   STATUS[239].EXT.Forced := FALSE;
   STATUS[239].EXT.BIT29 := FALSE;
   STATUS[239].EXT.BIT30 := FALSE;
   STATUS[239].EXT.BIT31 := FALSE;
   STATUS[239].EXT.ModeBit1 := FALSE;
   STATUS[239].EXT.ModeBit2 := FALSE;
   STATUS[239].EXT.ModeBit3 := FALSE;
   STATUS[239].EXT.BIT19 := FALSE;
   STATUS[239].EXT.BIT20 := FALSE;
   STATUS[239].EXT.AlarmSuppressed := FALSE;
   STATUS[239].EXT.AlarmPrsent := FALSE;
   STATUS[239].EXT.AlarmFailUnAck := FALSE;
   STATUS[239].Status := 0;
   STATUS[239].TimeStamp := 16#0000;
   STATUS[240].VALUE := 0.0;
   STATUS[240].TRIGVALUE := 0.0;
   STATUS[240].EXT.AlarmWarnUnAck := FALSE;
   STATUS[240].EXT.AckRequired := FALSE;
   STATUS[240].EXT.Maintanence := FALSE;
   STATUS[240].EXT.Operation := FALSE;
   STATUS[240].EXT.Forced := FALSE;
   STATUS[240].EXT.BIT29 := FALSE;
   STATUS[240].EXT.BIT30 := FALSE;
   STATUS[240].EXT.BIT31 := FALSE;
   STATUS[240].EXT.ModeBit1 := FALSE;
   STATUS[240].EXT.ModeBit2 := FALSE;
   STATUS[240].EXT.ModeBit3 := FALSE;
   STATUS[240].EXT.BIT19 := FALSE;
   STATUS[240].EXT.BIT20 := FALSE;
   STATUS[240].EXT.AlarmSuppressed := FALSE;
   STATUS[240].EXT.AlarmPrsent := FALSE;
   STATUS[240].EXT.AlarmFailUnAck := FALSE;
   STATUS[240].Status := 0;
   STATUS[240].TimeStamp := 16#0000;
   STATUS[241].VALUE := 0.0;
   STATUS[241].TRIGVALUE := 0.0;
   STATUS[241].EXT.AlarmWarnUnAck := FALSE;
   STATUS[241].EXT.AckRequired := FALSE;
   STATUS[241].EXT.Maintanence := FALSE;
   STATUS[241].EXT.Operation := FALSE;
   STATUS[241].EXT.Forced := FALSE;
   STATUS[241].EXT.BIT29 := FALSE;
   STATUS[241].EXT.BIT30 := FALSE;
   STATUS[241].EXT.BIT31 := FALSE;
   STATUS[241].EXT.ModeBit1 := FALSE;
   STATUS[241].EXT.ModeBit2 := FALSE;
   STATUS[241].EXT.ModeBit3 := FALSE;
   STATUS[241].EXT.BIT19 := FALSE;
   STATUS[241].EXT.BIT20 := FALSE;
   STATUS[241].EXT.AlarmSuppressed := FALSE;
   STATUS[241].EXT.AlarmPrsent := FALSE;
   STATUS[241].EXT.AlarmFailUnAck := FALSE;
   STATUS[241].Status := 0;
   STATUS[241].TimeStamp := 16#0000;
   STATUS[242].VALUE := 0.0;
   STATUS[242].TRIGVALUE := 0.0;
   STATUS[242].EXT.AlarmWarnUnAck := FALSE;
   STATUS[242].EXT.AckRequired := FALSE;
   STATUS[242].EXT.Maintanence := FALSE;
   STATUS[242].EXT.Operation := FALSE;
   STATUS[242].EXT.Forced := FALSE;
   STATUS[242].EXT.BIT29 := FALSE;
   STATUS[242].EXT.BIT30 := FALSE;
   STATUS[242].EXT.BIT31 := FALSE;
   STATUS[242].EXT.ModeBit1 := FALSE;
   STATUS[242].EXT.ModeBit2 := FALSE;
   STATUS[242].EXT.ModeBit3 := FALSE;
   STATUS[242].EXT.BIT19 := FALSE;
   STATUS[242].EXT.BIT20 := FALSE;
   STATUS[242].EXT.AlarmSuppressed := FALSE;
   STATUS[242].EXT.AlarmPrsent := FALSE;
   STATUS[242].EXT.AlarmFailUnAck := FALSE;
   STATUS[242].Status := 0;
   STATUS[242].TimeStamp := 16#0000;
   STATUS[243].VALUE := 0.0;
   STATUS[243].TRIGVALUE := 0.0;
   STATUS[243].EXT.AlarmWarnUnAck := FALSE;
   STATUS[243].EXT.AckRequired := FALSE;
   STATUS[243].EXT.Maintanence := FALSE;
   STATUS[243].EXT.Operation := FALSE;
   STATUS[243].EXT.Forced := FALSE;
   STATUS[243].EXT.BIT29 := FALSE;
   STATUS[243].EXT.BIT30 := FALSE;
   STATUS[243].EXT.BIT31 := FALSE;
   STATUS[243].EXT.ModeBit1 := FALSE;
   STATUS[243].EXT.ModeBit2 := FALSE;
   STATUS[243].EXT.ModeBit3 := FALSE;
   STATUS[243].EXT.BIT19 := FALSE;
   STATUS[243].EXT.BIT20 := FALSE;
   STATUS[243].EXT.AlarmSuppressed := FALSE;
   STATUS[243].EXT.AlarmPrsent := FALSE;
   STATUS[243].EXT.AlarmFailUnAck := FALSE;
   STATUS[243].Status := 0;
   STATUS[243].TimeStamp := 16#0000;
   STATUS[244].VALUE := 0.0;
   STATUS[244].TRIGVALUE := 0.0;
   STATUS[244].EXT.AlarmWarnUnAck := FALSE;
   STATUS[244].EXT.AckRequired := FALSE;
   STATUS[244].EXT.Maintanence := FALSE;
   STATUS[244].EXT.Operation := FALSE;
   STATUS[244].EXT.Forced := FALSE;
   STATUS[244].EXT.BIT29 := FALSE;
   STATUS[244].EXT.BIT30 := FALSE;
   STATUS[244].EXT.BIT31 := FALSE;
   STATUS[244].EXT.ModeBit1 := FALSE;
   STATUS[244].EXT.ModeBit2 := FALSE;
   STATUS[244].EXT.ModeBit3 := FALSE;
   STATUS[244].EXT.BIT19 := FALSE;
   STATUS[244].EXT.BIT20 := FALSE;
   STATUS[244].EXT.AlarmSuppressed := FALSE;
   STATUS[244].EXT.AlarmPrsent := FALSE;
   STATUS[244].EXT.AlarmFailUnAck := FALSE;
   STATUS[244].Status := 0;
   STATUS[244].TimeStamp := 16#0000;
   STATUS[245].VALUE := 0.0;
   STATUS[245].TRIGVALUE := 0.0;
   STATUS[245].EXT.AlarmWarnUnAck := FALSE;
   STATUS[245].EXT.AckRequired := FALSE;
   STATUS[245].EXT.Maintanence := FALSE;
   STATUS[245].EXT.Operation := FALSE;
   STATUS[245].EXT.Forced := FALSE;
   STATUS[245].EXT.BIT29 := FALSE;
   STATUS[245].EXT.BIT30 := FALSE;
   STATUS[245].EXT.BIT31 := FALSE;
   STATUS[245].EXT.ModeBit1 := FALSE;
   STATUS[245].EXT.ModeBit2 := FALSE;
   STATUS[245].EXT.ModeBit3 := FALSE;
   STATUS[245].EXT.BIT19 := FALSE;
   STATUS[245].EXT.BIT20 := FALSE;
   STATUS[245].EXT.AlarmSuppressed := FALSE;
   STATUS[245].EXT.AlarmPrsent := FALSE;
   STATUS[245].EXT.AlarmFailUnAck := FALSE;
   STATUS[245].Status := 0;
   STATUS[245].TimeStamp := 16#0000;
   STATUS[246].VALUE := 0.0;
   STATUS[246].TRIGVALUE := 0.0;
   STATUS[246].EXT.AlarmWarnUnAck := FALSE;
   STATUS[246].EXT.AckRequired := FALSE;
   STATUS[246].EXT.Maintanence := FALSE;
   STATUS[246].EXT.Operation := FALSE;
   STATUS[246].EXT.Forced := FALSE;
   STATUS[246].EXT.BIT29 := FALSE;
   STATUS[246].EXT.BIT30 := FALSE;
   STATUS[246].EXT.BIT31 := FALSE;
   STATUS[246].EXT.ModeBit1 := FALSE;
   STATUS[246].EXT.ModeBit2 := FALSE;
   STATUS[246].EXT.ModeBit3 := FALSE;
   STATUS[246].EXT.BIT19 := FALSE;
   STATUS[246].EXT.BIT20 := FALSE;
   STATUS[246].EXT.AlarmSuppressed := FALSE;
   STATUS[246].EXT.AlarmPrsent := FALSE;
   STATUS[246].EXT.AlarmFailUnAck := FALSE;
   STATUS[246].Status := 0;
   STATUS[246].TimeStamp := 16#0000;
   STATUS[247].VALUE := 0.0;
   STATUS[247].TRIGVALUE := 0.0;
   STATUS[247].EXT.AlarmWarnUnAck := FALSE;
   STATUS[247].EXT.AckRequired := FALSE;
   STATUS[247].EXT.Maintanence := FALSE;
   STATUS[247].EXT.Operation := FALSE;
   STATUS[247].EXT.Forced := FALSE;
   STATUS[247].EXT.BIT29 := FALSE;
   STATUS[247].EXT.BIT30 := FALSE;
   STATUS[247].EXT.BIT31 := FALSE;
   STATUS[247].EXT.ModeBit1 := FALSE;
   STATUS[247].EXT.ModeBit2 := FALSE;
   STATUS[247].EXT.ModeBit3 := FALSE;
   STATUS[247].EXT.BIT19 := FALSE;
   STATUS[247].EXT.BIT20 := FALSE;
   STATUS[247].EXT.AlarmSuppressed := FALSE;
   STATUS[247].EXT.AlarmPrsent := FALSE;
   STATUS[247].EXT.AlarmFailUnAck := FALSE;
   STATUS[247].Status := 0;
   STATUS[247].TimeStamp := 16#0000;
   STATUS[248].VALUE := 0.0;
   STATUS[248].TRIGVALUE := 0.0;
   STATUS[248].EXT.AlarmWarnUnAck := FALSE;
   STATUS[248].EXT.AckRequired := FALSE;
   STATUS[248].EXT.Maintanence := FALSE;
   STATUS[248].EXT.Operation := FALSE;
   STATUS[248].EXT.Forced := FALSE;
   STATUS[248].EXT.BIT29 := FALSE;
   STATUS[248].EXT.BIT30 := FALSE;
   STATUS[248].EXT.BIT31 := FALSE;
   STATUS[248].EXT.ModeBit1 := FALSE;
   STATUS[248].EXT.ModeBit2 := FALSE;
   STATUS[248].EXT.ModeBit3 := FALSE;
   STATUS[248].EXT.BIT19 := FALSE;
   STATUS[248].EXT.BIT20 := FALSE;
   STATUS[248].EXT.AlarmSuppressed := FALSE;
   STATUS[248].EXT.AlarmPrsent := FALSE;
   STATUS[248].EXT.AlarmFailUnAck := FALSE;
   STATUS[248].Status := 0;
   STATUS[248].TimeStamp := 16#0000;
   STATUS[249].VALUE := 0.0;
   STATUS[249].TRIGVALUE := 0.0;
   STATUS[249].EXT.AlarmWarnUnAck := FALSE;
   STATUS[249].EXT.AckRequired := FALSE;
   STATUS[249].EXT.Maintanence := FALSE;
   STATUS[249].EXT.Operation := FALSE;
   STATUS[249].EXT.Forced := FALSE;
   STATUS[249].EXT.BIT29 := FALSE;
   STATUS[249].EXT.BIT30 := FALSE;
   STATUS[249].EXT.BIT31 := FALSE;
   STATUS[249].EXT.ModeBit1 := FALSE;
   STATUS[249].EXT.ModeBit2 := FALSE;
   STATUS[249].EXT.ModeBit3 := FALSE;
   STATUS[249].EXT.BIT19 := FALSE;
   STATUS[249].EXT.BIT20 := FALSE;
   STATUS[249].EXT.AlarmSuppressed := FALSE;
   STATUS[249].EXT.AlarmPrsent := FALSE;
   STATUS[249].EXT.AlarmFailUnAck := FALSE;
   STATUS[249].Status := 0;
   STATUS[249].TimeStamp := 16#0000;
   STATUS[250].VALUE := 0.0;
   STATUS[250].TRIGVALUE := 0.0;
   STATUS[250].EXT.AlarmWarnUnAck := FALSE;
   STATUS[250].EXT.AckRequired := FALSE;
   STATUS[250].EXT.Maintanence := FALSE;
   STATUS[250].EXT.Operation := FALSE;
   STATUS[250].EXT.Forced := FALSE;
   STATUS[250].EXT.BIT29 := FALSE;
   STATUS[250].EXT.BIT30 := FALSE;
   STATUS[250].EXT.BIT31 := FALSE;
   STATUS[250].EXT.ModeBit1 := FALSE;
   STATUS[250].EXT.ModeBit2 := FALSE;
   STATUS[250].EXT.ModeBit3 := FALSE;
   STATUS[250].EXT.BIT19 := FALSE;
   STATUS[250].EXT.BIT20 := FALSE;
   STATUS[250].EXT.AlarmSuppressed := FALSE;
   STATUS[250].EXT.AlarmPrsent := FALSE;
   STATUS[250].EXT.AlarmFailUnAck := FALSE;
   STATUS[250].Status := 0;
   STATUS[250].TimeStamp := 16#0000;
   STATUS[251].VALUE := 0.0;
   STATUS[251].TRIGVALUE := 0.0;
   STATUS[251].EXT.AlarmWarnUnAck := FALSE;
   STATUS[251].EXT.AckRequired := FALSE;
   STATUS[251].EXT.Maintanence := FALSE;
   STATUS[251].EXT.Operation := FALSE;
   STATUS[251].EXT.Forced := FALSE;
   STATUS[251].EXT.BIT29 := FALSE;
   STATUS[251].EXT.BIT30 := FALSE;
   STATUS[251].EXT.BIT31 := FALSE;
   STATUS[251].EXT.ModeBit1 := FALSE;
   STATUS[251].EXT.ModeBit2 := FALSE;
   STATUS[251].EXT.ModeBit3 := FALSE;
   STATUS[251].EXT.BIT19 := FALSE;
   STATUS[251].EXT.BIT20 := FALSE;
   STATUS[251].EXT.AlarmSuppressed := FALSE;
   STATUS[251].EXT.AlarmPrsent := FALSE;
   STATUS[251].EXT.AlarmFailUnAck := FALSE;
   STATUS[251].Status := 0;
   STATUS[251].TimeStamp := 16#0000;
   STATUS[252].VALUE := 0.0;
   STATUS[252].TRIGVALUE := 0.0;
   STATUS[252].EXT.AlarmWarnUnAck := FALSE;
   STATUS[252].EXT.AckRequired := FALSE;
   STATUS[252].EXT.Maintanence := FALSE;
   STATUS[252].EXT.Operation := FALSE;
   STATUS[252].EXT.Forced := FALSE;
   STATUS[252].EXT.BIT29 := FALSE;
   STATUS[252].EXT.BIT30 := FALSE;
   STATUS[252].EXT.BIT31 := FALSE;
   STATUS[252].EXT.ModeBit1 := FALSE;
   STATUS[252].EXT.ModeBit2 := FALSE;
   STATUS[252].EXT.ModeBit3 := FALSE;
   STATUS[252].EXT.BIT19 := FALSE;
   STATUS[252].EXT.BIT20 := FALSE;
   STATUS[252].EXT.AlarmSuppressed := FALSE;
   STATUS[252].EXT.AlarmPrsent := FALSE;
   STATUS[252].EXT.AlarmFailUnAck := FALSE;
   STATUS[252].Status := 0;
   STATUS[252].TimeStamp := 16#0000;
   STATUS[253].VALUE := 0.0;
   STATUS[253].TRIGVALUE := 0.0;
   STATUS[253].EXT.AlarmWarnUnAck := FALSE;
   STATUS[253].EXT.AckRequired := FALSE;
   STATUS[253].EXT.Maintanence := FALSE;
   STATUS[253].EXT.Operation := FALSE;
   STATUS[253].EXT.Forced := FALSE;
   STATUS[253].EXT.BIT29 := FALSE;
   STATUS[253].EXT.BIT30 := FALSE;
   STATUS[253].EXT.BIT31 := FALSE;
   STATUS[253].EXT.ModeBit1 := FALSE;
   STATUS[253].EXT.ModeBit2 := FALSE;
   STATUS[253].EXT.ModeBit3 := FALSE;
   STATUS[253].EXT.BIT19 := FALSE;
   STATUS[253].EXT.BIT20 := FALSE;
   STATUS[253].EXT.AlarmSuppressed := FALSE;
   STATUS[253].EXT.AlarmPrsent := FALSE;
   STATUS[253].EXT.AlarmFailUnAck := FALSE;
   STATUS[253].Status := 0;
   STATUS[253].TimeStamp := 16#0000;
   STATUS[254].VALUE := 0.0;
   STATUS[254].TRIGVALUE := 0.0;
   STATUS[254].EXT.AlarmWarnUnAck := FALSE;
   STATUS[254].EXT.AckRequired := FALSE;
   STATUS[254].EXT.Maintanence := FALSE;
   STATUS[254].EXT.Operation := FALSE;
   STATUS[254].EXT.Forced := FALSE;
   STATUS[254].EXT.BIT29 := FALSE;
   STATUS[254].EXT.BIT30 := FALSE;
   STATUS[254].EXT.BIT31 := FALSE;
   STATUS[254].EXT.ModeBit1 := FALSE;
   STATUS[254].EXT.ModeBit2 := FALSE;
   STATUS[254].EXT.ModeBit3 := FALSE;
   STATUS[254].EXT.BIT19 := FALSE;
   STATUS[254].EXT.BIT20 := FALSE;
   STATUS[254].EXT.AlarmSuppressed := FALSE;
   STATUS[254].EXT.AlarmPrsent := FALSE;
   STATUS[254].EXT.AlarmFailUnAck := FALSE;
   STATUS[254].Status := 0;
   STATUS[254].TimeStamp := 16#0000;
   STATUS[255].VALUE := 0.0;
   STATUS[255].TRIGVALUE := 0.0;
   STATUS[255].EXT.AlarmWarnUnAck := FALSE;
   STATUS[255].EXT.AckRequired := FALSE;
   STATUS[255].EXT.Maintanence := FALSE;
   STATUS[255].EXT.Operation := FALSE;
   STATUS[255].EXT.Forced := FALSE;
   STATUS[255].EXT.BIT29 := FALSE;
   STATUS[255].EXT.BIT30 := FALSE;
   STATUS[255].EXT.BIT31 := FALSE;
   STATUS[255].EXT.ModeBit1 := FALSE;
   STATUS[255].EXT.ModeBit2 := FALSE;
   STATUS[255].EXT.ModeBit3 := FALSE;
   STATUS[255].EXT.BIT19 := FALSE;
   STATUS[255].EXT.BIT20 := FALSE;
   STATUS[255].EXT.AlarmSuppressed := FALSE;
   STATUS[255].EXT.AlarmPrsent := FALSE;
   STATUS[255].EXT.AlarmFailUnAck := FALSE;
   STATUS[255].Status := 0;
   STATUS[255].TimeStamp := 16#0000;
   STATUS[256].VALUE := 0.0;
   STATUS[256].TRIGVALUE := 0.0;
   STATUS[256].EXT.AlarmWarnUnAck := FALSE;
   STATUS[256].EXT.AckRequired := FALSE;
   STATUS[256].EXT.Maintanence := FALSE;
   STATUS[256].EXT.Operation := FALSE;
   STATUS[256].EXT.Forced := FALSE;
   STATUS[256].EXT.BIT29 := FALSE;
   STATUS[256].EXT.BIT30 := FALSE;
   STATUS[256].EXT.BIT31 := FALSE;
   STATUS[256].EXT.ModeBit1 := FALSE;
   STATUS[256].EXT.ModeBit2 := FALSE;
   STATUS[256].EXT.ModeBit3 := FALSE;
   STATUS[256].EXT.BIT19 := FALSE;
   STATUS[256].EXT.BIT20 := FALSE;
   STATUS[256].EXT.AlarmSuppressed := FALSE;
   STATUS[256].EXT.AlarmPrsent := FALSE;
   STATUS[256].EXT.AlarmFailUnAck := FALSE;
   STATUS[256].Status := 0;
   STATUS[256].TimeStamp := 16#0000;
   STATUS[257].VALUE := 0.0;
   STATUS[257].TRIGVALUE := 0.0;
   STATUS[257].EXT.AlarmWarnUnAck := FALSE;
   STATUS[257].EXT.AckRequired := FALSE;
   STATUS[257].EXT.Maintanence := FALSE;
   STATUS[257].EXT.Operation := FALSE;
   STATUS[257].EXT.Forced := FALSE;
   STATUS[257].EXT.BIT29 := FALSE;
   STATUS[257].EXT.BIT30 := FALSE;
   STATUS[257].EXT.BIT31 := FALSE;
   STATUS[257].EXT.ModeBit1 := FALSE;
   STATUS[257].EXT.ModeBit2 := FALSE;
   STATUS[257].EXT.ModeBit3 := FALSE;
   STATUS[257].EXT.BIT19 := FALSE;
   STATUS[257].EXT.BIT20 := FALSE;
   STATUS[257].EXT.AlarmSuppressed := FALSE;
   STATUS[257].EXT.AlarmPrsent := FALSE;
   STATUS[257].EXT.AlarmFailUnAck := FALSE;
   STATUS[257].Status := 0;
   STATUS[257].TimeStamp := 16#0000;
   STATUS[258].VALUE := 0.0;
   STATUS[258].TRIGVALUE := 0.0;
   STATUS[258].EXT.AlarmWarnUnAck := FALSE;
   STATUS[258].EXT.AckRequired := FALSE;
   STATUS[258].EXT.Maintanence := FALSE;
   STATUS[258].EXT.Operation := FALSE;
   STATUS[258].EXT.Forced := FALSE;
   STATUS[258].EXT.BIT29 := FALSE;
   STATUS[258].EXT.BIT30 := FALSE;
   STATUS[258].EXT.BIT31 := FALSE;
   STATUS[258].EXT.ModeBit1 := FALSE;
   STATUS[258].EXT.ModeBit2 := FALSE;
   STATUS[258].EXT.ModeBit3 := FALSE;
   STATUS[258].EXT.BIT19 := FALSE;
   STATUS[258].EXT.BIT20 := FALSE;
   STATUS[258].EXT.AlarmSuppressed := FALSE;
   STATUS[258].EXT.AlarmPrsent := FALSE;
   STATUS[258].EXT.AlarmFailUnAck := FALSE;
   STATUS[258].Status := 0;
   STATUS[258].TimeStamp := 16#0000;
   STATUS[259].VALUE := 0.0;
   STATUS[259].TRIGVALUE := 0.0;
   STATUS[259].EXT.AlarmWarnUnAck := FALSE;
   STATUS[259].EXT.AckRequired := FALSE;
   STATUS[259].EXT.Maintanence := FALSE;
   STATUS[259].EXT.Operation := FALSE;
   STATUS[259].EXT.Forced := FALSE;
   STATUS[259].EXT.BIT29 := FALSE;
   STATUS[259].EXT.BIT30 := FALSE;
   STATUS[259].EXT.BIT31 := FALSE;
   STATUS[259].EXT.ModeBit1 := FALSE;
   STATUS[259].EXT.ModeBit2 := FALSE;
   STATUS[259].EXT.ModeBit3 := FALSE;
   STATUS[259].EXT.BIT19 := FALSE;
   STATUS[259].EXT.BIT20 := FALSE;
   STATUS[259].EXT.AlarmSuppressed := FALSE;
   STATUS[259].EXT.AlarmPrsent := FALSE;
   STATUS[259].EXT.AlarmFailUnAck := FALSE;
   STATUS[259].Status := 0;
   STATUS[259].TimeStamp := 16#0000;
   STATUS[260].VALUE := 0.0;
   STATUS[260].TRIGVALUE := 0.0;
   STATUS[260].EXT.AlarmWarnUnAck := FALSE;
   STATUS[260].EXT.AckRequired := FALSE;
   STATUS[260].EXT.Maintanence := FALSE;
   STATUS[260].EXT.Operation := FALSE;
   STATUS[260].EXT.Forced := FALSE;
   STATUS[260].EXT.BIT29 := FALSE;
   STATUS[260].EXT.BIT30 := FALSE;
   STATUS[260].EXT.BIT31 := FALSE;
   STATUS[260].EXT.ModeBit1 := FALSE;
   STATUS[260].EXT.ModeBit2 := FALSE;
   STATUS[260].EXT.ModeBit3 := FALSE;
   STATUS[260].EXT.BIT19 := FALSE;
   STATUS[260].EXT.BIT20 := FALSE;
   STATUS[260].EXT.AlarmSuppressed := FALSE;
   STATUS[260].EXT.AlarmPrsent := FALSE;
   STATUS[260].EXT.AlarmFailUnAck := FALSE;
   STATUS[260].Status := 0;
   STATUS[260].TimeStamp := 16#0000;
   STATUS[261].VALUE := 0.0;
   STATUS[261].TRIGVALUE := 0.0;
   STATUS[261].EXT.AlarmWarnUnAck := FALSE;
   STATUS[261].EXT.AckRequired := FALSE;
   STATUS[261].EXT.Maintanence := FALSE;
   STATUS[261].EXT.Operation := FALSE;
   STATUS[261].EXT.Forced := FALSE;
   STATUS[261].EXT.BIT29 := FALSE;
   STATUS[261].EXT.BIT30 := FALSE;
   STATUS[261].EXT.BIT31 := FALSE;
   STATUS[261].EXT.ModeBit1 := FALSE;
   STATUS[261].EXT.ModeBit2 := FALSE;
   STATUS[261].EXT.ModeBit3 := FALSE;
   STATUS[261].EXT.BIT19 := FALSE;
   STATUS[261].EXT.BIT20 := FALSE;
   STATUS[261].EXT.AlarmSuppressed := FALSE;
   STATUS[261].EXT.AlarmPrsent := FALSE;
   STATUS[261].EXT.AlarmFailUnAck := FALSE;
   STATUS[261].Status := 0;
   STATUS[261].TimeStamp := 16#0000;
   STATUS[262].VALUE := 0.0;
   STATUS[262].TRIGVALUE := 0.0;
   STATUS[262].EXT.AlarmWarnUnAck := FALSE;
   STATUS[262].EXT.AckRequired := FALSE;
   STATUS[262].EXT.Maintanence := FALSE;
   STATUS[262].EXT.Operation := FALSE;
   STATUS[262].EXT.Forced := FALSE;
   STATUS[262].EXT.BIT29 := FALSE;
   STATUS[262].EXT.BIT30 := FALSE;
   STATUS[262].EXT.BIT31 := FALSE;
   STATUS[262].EXT.ModeBit1 := FALSE;
   STATUS[262].EXT.ModeBit2 := FALSE;
   STATUS[262].EXT.ModeBit3 := FALSE;
   STATUS[262].EXT.BIT19 := FALSE;
   STATUS[262].EXT.BIT20 := FALSE;
   STATUS[262].EXT.AlarmSuppressed := FALSE;
   STATUS[262].EXT.AlarmPrsent := FALSE;
   STATUS[262].EXT.AlarmFailUnAck := FALSE;
   STATUS[262].Status := 0;
   STATUS[262].TimeStamp := 16#0000;
   STATUS[263].VALUE := 0.0;
   STATUS[263].TRIGVALUE := 0.0;
   STATUS[263].EXT.AlarmWarnUnAck := FALSE;
   STATUS[263].EXT.AckRequired := FALSE;
   STATUS[263].EXT.Maintanence := FALSE;
   STATUS[263].EXT.Operation := FALSE;
   STATUS[263].EXT.Forced := FALSE;
   STATUS[263].EXT.BIT29 := FALSE;
   STATUS[263].EXT.BIT30 := FALSE;
   STATUS[263].EXT.BIT31 := FALSE;
   STATUS[263].EXT.ModeBit1 := FALSE;
   STATUS[263].EXT.ModeBit2 := FALSE;
   STATUS[263].EXT.ModeBit3 := FALSE;
   STATUS[263].EXT.BIT19 := FALSE;
   STATUS[263].EXT.BIT20 := FALSE;
   STATUS[263].EXT.AlarmSuppressed := FALSE;
   STATUS[263].EXT.AlarmPrsent := FALSE;
   STATUS[263].EXT.AlarmFailUnAck := FALSE;
   STATUS[263].Status := 0;
   STATUS[263].TimeStamp := 16#0000;
   STATUS[264].VALUE := 0.0;
   STATUS[264].TRIGVALUE := 0.0;
   STATUS[264].EXT.AlarmWarnUnAck := FALSE;
   STATUS[264].EXT.AckRequired := FALSE;
   STATUS[264].EXT.Maintanence := FALSE;
   STATUS[264].EXT.Operation := FALSE;
   STATUS[264].EXT.Forced := FALSE;
   STATUS[264].EXT.BIT29 := FALSE;
   STATUS[264].EXT.BIT30 := FALSE;
   STATUS[264].EXT.BIT31 := FALSE;
   STATUS[264].EXT.ModeBit1 := FALSE;
   STATUS[264].EXT.ModeBit2 := FALSE;
   STATUS[264].EXT.ModeBit3 := FALSE;
   STATUS[264].EXT.BIT19 := FALSE;
   STATUS[264].EXT.BIT20 := FALSE;
   STATUS[264].EXT.AlarmSuppressed := FALSE;
   STATUS[264].EXT.AlarmPrsent := FALSE;
   STATUS[264].EXT.AlarmFailUnAck := FALSE;
   STATUS[264].Status := 0;
   STATUS[264].TimeStamp := 16#0000;
   STATUS[265].VALUE := 0.0;
   STATUS[265].TRIGVALUE := 0.0;
   STATUS[265].EXT.AlarmWarnUnAck := FALSE;
   STATUS[265].EXT.AckRequired := FALSE;
   STATUS[265].EXT.Maintanence := FALSE;
   STATUS[265].EXT.Operation := FALSE;
   STATUS[265].EXT.Forced := FALSE;
   STATUS[265].EXT.BIT29 := FALSE;
   STATUS[265].EXT.BIT30 := FALSE;
   STATUS[265].EXT.BIT31 := FALSE;
   STATUS[265].EXT.ModeBit1 := FALSE;
   STATUS[265].EXT.ModeBit2 := FALSE;
   STATUS[265].EXT.ModeBit3 := FALSE;
   STATUS[265].EXT.BIT19 := FALSE;
   STATUS[265].EXT.BIT20 := FALSE;
   STATUS[265].EXT.AlarmSuppressed := FALSE;
   STATUS[265].EXT.AlarmPrsent := FALSE;
   STATUS[265].EXT.AlarmFailUnAck := FALSE;
   STATUS[265].Status := 0;
   STATUS[265].TimeStamp := 16#0000;
   STATUS[266].VALUE := 0.0;
   STATUS[266].TRIGVALUE := 0.0;
   STATUS[266].EXT.AlarmWarnUnAck := FALSE;
   STATUS[266].EXT.AckRequired := FALSE;
   STATUS[266].EXT.Maintanence := FALSE;
   STATUS[266].EXT.Operation := FALSE;
   STATUS[266].EXT.Forced := FALSE;
   STATUS[266].EXT.BIT29 := FALSE;
   STATUS[266].EXT.BIT30 := FALSE;
   STATUS[266].EXT.BIT31 := FALSE;
   STATUS[266].EXT.ModeBit1 := FALSE;
   STATUS[266].EXT.ModeBit2 := FALSE;
   STATUS[266].EXT.ModeBit3 := FALSE;
   STATUS[266].EXT.BIT19 := FALSE;
   STATUS[266].EXT.BIT20 := FALSE;
   STATUS[266].EXT.AlarmSuppressed := FALSE;
   STATUS[266].EXT.AlarmPrsent := FALSE;
   STATUS[266].EXT.AlarmFailUnAck := FALSE;
   STATUS[266].Status := 0;
   STATUS[266].TimeStamp := 16#0000;
   STATUS[267].VALUE := 0.0;
   STATUS[267].TRIGVALUE := 0.0;
   STATUS[267].EXT.AlarmWarnUnAck := FALSE;
   STATUS[267].EXT.AckRequired := FALSE;
   STATUS[267].EXT.Maintanence := FALSE;
   STATUS[267].EXT.Operation := FALSE;
   STATUS[267].EXT.Forced := FALSE;
   STATUS[267].EXT.BIT29 := FALSE;
   STATUS[267].EXT.BIT30 := FALSE;
   STATUS[267].EXT.BIT31 := FALSE;
   STATUS[267].EXT.ModeBit1 := FALSE;
   STATUS[267].EXT.ModeBit2 := FALSE;
   STATUS[267].EXT.ModeBit3 := FALSE;
   STATUS[267].EXT.BIT19 := FALSE;
   STATUS[267].EXT.BIT20 := FALSE;
   STATUS[267].EXT.AlarmSuppressed := FALSE;
   STATUS[267].EXT.AlarmPrsent := FALSE;
   STATUS[267].EXT.AlarmFailUnAck := FALSE;
   STATUS[267].Status := 0;
   STATUS[267].TimeStamp := 16#0000;
   STATUS[268].VALUE := 0.0;
   STATUS[268].TRIGVALUE := 0.0;
   STATUS[268].EXT.AlarmWarnUnAck := FALSE;
   STATUS[268].EXT.AckRequired := FALSE;
   STATUS[268].EXT.Maintanence := FALSE;
   STATUS[268].EXT.Operation := FALSE;
   STATUS[268].EXT.Forced := FALSE;
   STATUS[268].EXT.BIT29 := FALSE;
   STATUS[268].EXT.BIT30 := FALSE;
   STATUS[268].EXT.BIT31 := FALSE;
   STATUS[268].EXT.ModeBit1 := FALSE;
   STATUS[268].EXT.ModeBit2 := FALSE;
   STATUS[268].EXT.ModeBit3 := FALSE;
   STATUS[268].EXT.BIT19 := FALSE;
   STATUS[268].EXT.BIT20 := FALSE;
   STATUS[268].EXT.AlarmSuppressed := FALSE;
   STATUS[268].EXT.AlarmPrsent := FALSE;
   STATUS[268].EXT.AlarmFailUnAck := FALSE;
   STATUS[268].Status := 0;
   STATUS[268].TimeStamp := 16#0000;
   STATUS[269].VALUE := 0.0;
   STATUS[269].TRIGVALUE := 0.0;
   STATUS[269].EXT.AlarmWarnUnAck := FALSE;
   STATUS[269].EXT.AckRequired := FALSE;
   STATUS[269].EXT.Maintanence := FALSE;
   STATUS[269].EXT.Operation := FALSE;
   STATUS[269].EXT.Forced := FALSE;
   STATUS[269].EXT.BIT29 := FALSE;
   STATUS[269].EXT.BIT30 := FALSE;
   STATUS[269].EXT.BIT31 := FALSE;
   STATUS[269].EXT.ModeBit1 := FALSE;
   STATUS[269].EXT.ModeBit2 := FALSE;
   STATUS[269].EXT.ModeBit3 := FALSE;
   STATUS[269].EXT.BIT19 := FALSE;
   STATUS[269].EXT.BIT20 := FALSE;
   STATUS[269].EXT.AlarmSuppressed := FALSE;
   STATUS[269].EXT.AlarmPrsent := FALSE;
   STATUS[269].EXT.AlarmFailUnAck := FALSE;
   STATUS[269].Status := 0;
   STATUS[269].TimeStamp := 16#0000;
   STATUS[270].VALUE := 0.0;
   STATUS[270].TRIGVALUE := 0.0;
   STATUS[270].EXT.AlarmWarnUnAck := FALSE;
   STATUS[270].EXT.AckRequired := FALSE;
   STATUS[270].EXT.Maintanence := FALSE;
   STATUS[270].EXT.Operation := FALSE;
   STATUS[270].EXT.Forced := FALSE;
   STATUS[270].EXT.BIT29 := FALSE;
   STATUS[270].EXT.BIT30 := FALSE;
   STATUS[270].EXT.BIT31 := FALSE;
   STATUS[270].EXT.ModeBit1 := FALSE;
   STATUS[270].EXT.ModeBit2 := FALSE;
   STATUS[270].EXT.ModeBit3 := FALSE;
   STATUS[270].EXT.BIT19 := FALSE;
   STATUS[270].EXT.BIT20 := FALSE;
   STATUS[270].EXT.AlarmSuppressed := FALSE;
   STATUS[270].EXT.AlarmPrsent := FALSE;
   STATUS[270].EXT.AlarmFailUnAck := FALSE;
   STATUS[270].Status := 0;
   STATUS[270].TimeStamp := 16#0000;
   STATUS[271].VALUE := 0.0;
   STATUS[271].TRIGVALUE := 0.0;
   STATUS[271].EXT.AlarmWarnUnAck := FALSE;
   STATUS[271].EXT.AckRequired := FALSE;
   STATUS[271].EXT.Maintanence := FALSE;
   STATUS[271].EXT.Operation := FALSE;
   STATUS[271].EXT.Forced := FALSE;
   STATUS[271].EXT.BIT29 := FALSE;
   STATUS[271].EXT.BIT30 := FALSE;
   STATUS[271].EXT.BIT31 := FALSE;
   STATUS[271].EXT.ModeBit1 := FALSE;
   STATUS[271].EXT.ModeBit2 := FALSE;
   STATUS[271].EXT.ModeBit3 := FALSE;
   STATUS[271].EXT.BIT19 := FALSE;
   STATUS[271].EXT.BIT20 := FALSE;
   STATUS[271].EXT.AlarmSuppressed := FALSE;
   STATUS[271].EXT.AlarmPrsent := FALSE;
   STATUS[271].EXT.AlarmFailUnAck := FALSE;
   STATUS[271].Status := 0;
   STATUS[271].TimeStamp := 16#0000;
   STATUS[272].VALUE := 0.0;
   STATUS[272].TRIGVALUE := 0.0;
   STATUS[272].EXT.AlarmWarnUnAck := FALSE;
   STATUS[272].EXT.AckRequired := FALSE;
   STATUS[272].EXT.Maintanence := FALSE;
   STATUS[272].EXT.Operation := FALSE;
   STATUS[272].EXT.Forced := FALSE;
   STATUS[272].EXT.BIT29 := FALSE;
   STATUS[272].EXT.BIT30 := FALSE;
   STATUS[272].EXT.BIT31 := FALSE;
   STATUS[272].EXT.ModeBit1 := FALSE;
   STATUS[272].EXT.ModeBit2 := FALSE;
   STATUS[272].EXT.ModeBit3 := FALSE;
   STATUS[272].EXT.BIT19 := FALSE;
   STATUS[272].EXT.BIT20 := FALSE;
   STATUS[272].EXT.AlarmSuppressed := FALSE;
   STATUS[272].EXT.AlarmPrsent := FALSE;
   STATUS[272].EXT.AlarmFailUnAck := FALSE;
   STATUS[272].Status := 0;
   STATUS[272].TimeStamp := 16#0000;
   STATUS[273].VALUE := 0.0;
   STATUS[273].TRIGVALUE := 0.0;
   STATUS[273].EXT.AlarmWarnUnAck := FALSE;
   STATUS[273].EXT.AckRequired := FALSE;
   STATUS[273].EXT.Maintanence := FALSE;
   STATUS[273].EXT.Operation := FALSE;
   STATUS[273].EXT.Forced := FALSE;
   STATUS[273].EXT.BIT29 := FALSE;
   STATUS[273].EXT.BIT30 := FALSE;
   STATUS[273].EXT.BIT31 := FALSE;
   STATUS[273].EXT.ModeBit1 := FALSE;
   STATUS[273].EXT.ModeBit2 := FALSE;
   STATUS[273].EXT.ModeBit3 := FALSE;
   STATUS[273].EXT.BIT19 := FALSE;
   STATUS[273].EXT.BIT20 := FALSE;
   STATUS[273].EXT.AlarmSuppressed := FALSE;
   STATUS[273].EXT.AlarmPrsent := FALSE;
   STATUS[273].EXT.AlarmFailUnAck := FALSE;
   STATUS[273].Status := 0;
   STATUS[273].TimeStamp := 16#0000;
   STATUS[274].VALUE := 0.0;
   STATUS[274].TRIGVALUE := 0.0;
   STATUS[274].EXT.AlarmWarnUnAck := FALSE;
   STATUS[274].EXT.AckRequired := FALSE;
   STATUS[274].EXT.Maintanence := FALSE;
   STATUS[274].EXT.Operation := FALSE;
   STATUS[274].EXT.Forced := FALSE;
   STATUS[274].EXT.BIT29 := FALSE;
   STATUS[274].EXT.BIT30 := FALSE;
   STATUS[274].EXT.BIT31 := FALSE;
   STATUS[274].EXT.ModeBit1 := FALSE;
   STATUS[274].EXT.ModeBit2 := FALSE;
   STATUS[274].EXT.ModeBit3 := FALSE;
   STATUS[274].EXT.BIT19 := FALSE;
   STATUS[274].EXT.BIT20 := FALSE;
   STATUS[274].EXT.AlarmSuppressed := FALSE;
   STATUS[274].EXT.AlarmPrsent := FALSE;
   STATUS[274].EXT.AlarmFailUnAck := FALSE;
   STATUS[274].Status := 0;
   STATUS[274].TimeStamp := 16#0000;
   STATUS[275].VALUE := 0.0;
   STATUS[275].TRIGVALUE := 0.0;
   STATUS[275].EXT.AlarmWarnUnAck := FALSE;
   STATUS[275].EXT.AckRequired := FALSE;
   STATUS[275].EXT.Maintanence := FALSE;
   STATUS[275].EXT.Operation := FALSE;
   STATUS[275].EXT.Forced := FALSE;
   STATUS[275].EXT.BIT29 := FALSE;
   STATUS[275].EXT.BIT30 := FALSE;
   STATUS[275].EXT.BIT31 := FALSE;
   STATUS[275].EXT.ModeBit1 := FALSE;
   STATUS[275].EXT.ModeBit2 := FALSE;
   STATUS[275].EXT.ModeBit3 := FALSE;
   STATUS[275].EXT.BIT19 := FALSE;
   STATUS[275].EXT.BIT20 := FALSE;
   STATUS[275].EXT.AlarmSuppressed := FALSE;
   STATUS[275].EXT.AlarmPrsent := FALSE;
   STATUS[275].EXT.AlarmFailUnAck := FALSE;
   STATUS[275].Status := 0;
   STATUS[275].TimeStamp := 16#0000;
   STATUS[276].VALUE := 0.0;
   STATUS[276].TRIGVALUE := 0.0;
   STATUS[276].EXT.AlarmWarnUnAck := FALSE;
   STATUS[276].EXT.AckRequired := FALSE;
   STATUS[276].EXT.Maintanence := FALSE;
   STATUS[276].EXT.Operation := FALSE;
   STATUS[276].EXT.Forced := FALSE;
   STATUS[276].EXT.BIT29 := FALSE;
   STATUS[276].EXT.BIT30 := FALSE;
   STATUS[276].EXT.BIT31 := FALSE;
   STATUS[276].EXT.ModeBit1 := FALSE;
   STATUS[276].EXT.ModeBit2 := FALSE;
   STATUS[276].EXT.ModeBit3 := FALSE;
   STATUS[276].EXT.BIT19 := FALSE;
   STATUS[276].EXT.BIT20 := FALSE;
   STATUS[276].EXT.AlarmSuppressed := FALSE;
   STATUS[276].EXT.AlarmPrsent := FALSE;
   STATUS[276].EXT.AlarmFailUnAck := FALSE;
   STATUS[276].Status := 0;
   STATUS[276].TimeStamp := 16#0000;
   STATUS[277].VALUE := 0.0;
   STATUS[277].TRIGVALUE := 0.0;
   STATUS[277].EXT.AlarmWarnUnAck := FALSE;
   STATUS[277].EXT.AckRequired := FALSE;
   STATUS[277].EXT.Maintanence := FALSE;
   STATUS[277].EXT.Operation := FALSE;
   STATUS[277].EXT.Forced := FALSE;
   STATUS[277].EXT.BIT29 := FALSE;
   STATUS[277].EXT.BIT30 := FALSE;
   STATUS[277].EXT.BIT31 := FALSE;
   STATUS[277].EXT.ModeBit1 := FALSE;
   STATUS[277].EXT.ModeBit2 := FALSE;
   STATUS[277].EXT.ModeBit3 := FALSE;
   STATUS[277].EXT.BIT19 := FALSE;
   STATUS[277].EXT.BIT20 := FALSE;
   STATUS[277].EXT.AlarmSuppressed := FALSE;
   STATUS[277].EXT.AlarmPrsent := FALSE;
   STATUS[277].EXT.AlarmFailUnAck := FALSE;
   STATUS[277].Status := 0;
   STATUS[277].TimeStamp := 16#0000;
   STATUS[278].VALUE := 0.0;
   STATUS[278].TRIGVALUE := 0.0;
   STATUS[278].EXT.AlarmWarnUnAck := FALSE;
   STATUS[278].EXT.AckRequired := FALSE;
   STATUS[278].EXT.Maintanence := FALSE;
   STATUS[278].EXT.Operation := FALSE;
   STATUS[278].EXT.Forced := FALSE;
   STATUS[278].EXT.BIT29 := FALSE;
   STATUS[278].EXT.BIT30 := FALSE;
   STATUS[278].EXT.BIT31 := FALSE;
   STATUS[278].EXT.ModeBit1 := FALSE;
   STATUS[278].EXT.ModeBit2 := FALSE;
   STATUS[278].EXT.ModeBit3 := FALSE;
   STATUS[278].EXT.BIT19 := FALSE;
   STATUS[278].EXT.BIT20 := FALSE;
   STATUS[278].EXT.AlarmSuppressed := FALSE;
   STATUS[278].EXT.AlarmPrsent := FALSE;
   STATUS[278].EXT.AlarmFailUnAck := FALSE;
   STATUS[278].Status := 0;
   STATUS[278].TimeStamp := 16#0000;
   STATUS[279].VALUE := 0.0;
   STATUS[279].TRIGVALUE := 0.0;
   STATUS[279].EXT.AlarmWarnUnAck := FALSE;
   STATUS[279].EXT.AckRequired := FALSE;
   STATUS[279].EXT.Maintanence := FALSE;
   STATUS[279].EXT.Operation := FALSE;
   STATUS[279].EXT.Forced := FALSE;
   STATUS[279].EXT.BIT29 := FALSE;
   STATUS[279].EXT.BIT30 := FALSE;
   STATUS[279].EXT.BIT31 := FALSE;
   STATUS[279].EXT.ModeBit1 := FALSE;
   STATUS[279].EXT.ModeBit2 := FALSE;
   STATUS[279].EXT.ModeBit3 := FALSE;
   STATUS[279].EXT.BIT19 := FALSE;
   STATUS[279].EXT.BIT20 := FALSE;
   STATUS[279].EXT.AlarmSuppressed := FALSE;
   STATUS[279].EXT.AlarmPrsent := FALSE;
   STATUS[279].EXT.AlarmFailUnAck := FALSE;
   STATUS[279].Status := 0;
   STATUS[279].TimeStamp := 16#0000;
   STATUS[280].VALUE := 0.0;
   STATUS[280].TRIGVALUE := 0.0;
   STATUS[280].EXT.AlarmWarnUnAck := FALSE;
   STATUS[280].EXT.AckRequired := FALSE;
   STATUS[280].EXT.Maintanence := FALSE;
   STATUS[280].EXT.Operation := FALSE;
   STATUS[280].EXT.Forced := FALSE;
   STATUS[280].EXT.BIT29 := FALSE;
   STATUS[280].EXT.BIT30 := FALSE;
   STATUS[280].EXT.BIT31 := FALSE;
   STATUS[280].EXT.ModeBit1 := FALSE;
   STATUS[280].EXT.ModeBit2 := FALSE;
   STATUS[280].EXT.ModeBit3 := FALSE;
   STATUS[280].EXT.BIT19 := FALSE;
   STATUS[280].EXT.BIT20 := FALSE;
   STATUS[280].EXT.AlarmSuppressed := FALSE;
   STATUS[280].EXT.AlarmPrsent := FALSE;
   STATUS[280].EXT.AlarmFailUnAck := FALSE;
   STATUS[280].Status := 0;
   STATUS[280].TimeStamp := 16#0000;
   STATUS[281].VALUE := 0.0;
   STATUS[281].TRIGVALUE := 0.0;
   STATUS[281].EXT.AlarmWarnUnAck := FALSE;
   STATUS[281].EXT.AckRequired := FALSE;
   STATUS[281].EXT.Maintanence := FALSE;
   STATUS[281].EXT.Operation := FALSE;
   STATUS[281].EXT.Forced := FALSE;
   STATUS[281].EXT.BIT29 := FALSE;
   STATUS[281].EXT.BIT30 := FALSE;
   STATUS[281].EXT.BIT31 := FALSE;
   STATUS[281].EXT.ModeBit1 := FALSE;
   STATUS[281].EXT.ModeBit2 := FALSE;
   STATUS[281].EXT.ModeBit3 := FALSE;
   STATUS[281].EXT.BIT19 := FALSE;
   STATUS[281].EXT.BIT20 := FALSE;
   STATUS[281].EXT.AlarmSuppressed := FALSE;
   STATUS[281].EXT.AlarmPrsent := FALSE;
   STATUS[281].EXT.AlarmFailUnAck := FALSE;
   STATUS[281].Status := 0;
   STATUS[281].TimeStamp := 16#0000;
   STATUS[282].VALUE := 0.0;
   STATUS[282].TRIGVALUE := 0.0;
   STATUS[282].EXT.AlarmWarnUnAck := FALSE;
   STATUS[282].EXT.AckRequired := FALSE;
   STATUS[282].EXT.Maintanence := FALSE;
   STATUS[282].EXT.Operation := FALSE;
   STATUS[282].EXT.Forced := FALSE;
   STATUS[282].EXT.BIT29 := FALSE;
   STATUS[282].EXT.BIT30 := FALSE;
   STATUS[282].EXT.BIT31 := FALSE;
   STATUS[282].EXT.ModeBit1 := FALSE;
   STATUS[282].EXT.ModeBit2 := FALSE;
   STATUS[282].EXT.ModeBit3 := FALSE;
   STATUS[282].EXT.BIT19 := FALSE;
   STATUS[282].EXT.BIT20 := FALSE;
   STATUS[282].EXT.AlarmSuppressed := FALSE;
   STATUS[282].EXT.AlarmPrsent := FALSE;
   STATUS[282].EXT.AlarmFailUnAck := FALSE;
   STATUS[282].Status := 0;
   STATUS[282].TimeStamp := 16#0000;
   STATUS[283].VALUE := 0.0;
   STATUS[283].TRIGVALUE := 0.0;
   STATUS[283].EXT.AlarmWarnUnAck := FALSE;
   STATUS[283].EXT.AckRequired := FALSE;
   STATUS[283].EXT.Maintanence := FALSE;
   STATUS[283].EXT.Operation := FALSE;
   STATUS[283].EXT.Forced := FALSE;
   STATUS[283].EXT.BIT29 := FALSE;
   STATUS[283].EXT.BIT30 := FALSE;
   STATUS[283].EXT.BIT31 := FALSE;
   STATUS[283].EXT.ModeBit1 := FALSE;
   STATUS[283].EXT.ModeBit2 := FALSE;
   STATUS[283].EXT.ModeBit3 := FALSE;
   STATUS[283].EXT.BIT19 := FALSE;
   STATUS[283].EXT.BIT20 := FALSE;
   STATUS[283].EXT.AlarmSuppressed := FALSE;
   STATUS[283].EXT.AlarmPrsent := FALSE;
   STATUS[283].EXT.AlarmFailUnAck := FALSE;
   STATUS[283].Status := 0;
   STATUS[283].TimeStamp := 16#0000;
   STATUS[284].VALUE := 0.0;
   STATUS[284].TRIGVALUE := 0.0;
   STATUS[284].EXT.AlarmWarnUnAck := FALSE;
   STATUS[284].EXT.AckRequired := FALSE;
   STATUS[284].EXT.Maintanence := FALSE;
   STATUS[284].EXT.Operation := FALSE;
   STATUS[284].EXT.Forced := FALSE;
   STATUS[284].EXT.BIT29 := FALSE;
   STATUS[284].EXT.BIT30 := FALSE;
   STATUS[284].EXT.BIT31 := FALSE;
   STATUS[284].EXT.ModeBit1 := FALSE;
   STATUS[284].EXT.ModeBit2 := FALSE;
   STATUS[284].EXT.ModeBit3 := FALSE;
   STATUS[284].EXT.BIT19 := FALSE;
   STATUS[284].EXT.BIT20 := FALSE;
   STATUS[284].EXT.AlarmSuppressed := FALSE;
   STATUS[284].EXT.AlarmPrsent := FALSE;
   STATUS[284].EXT.AlarmFailUnAck := FALSE;
   STATUS[284].Status := 0;
   STATUS[284].TimeStamp := 16#0000;
   STATUS[285].VALUE := 0.0;
   STATUS[285].TRIGVALUE := 0.0;
   STATUS[285].EXT.AlarmWarnUnAck := FALSE;
   STATUS[285].EXT.AckRequired := FALSE;
   STATUS[285].EXT.Maintanence := FALSE;
   STATUS[285].EXT.Operation := FALSE;
   STATUS[285].EXT.Forced := FALSE;
   STATUS[285].EXT.BIT29 := FALSE;
   STATUS[285].EXT.BIT30 := FALSE;
   STATUS[285].EXT.BIT31 := FALSE;
   STATUS[285].EXT.ModeBit1 := FALSE;
   STATUS[285].EXT.ModeBit2 := FALSE;
   STATUS[285].EXT.ModeBit3 := FALSE;
   STATUS[285].EXT.BIT19 := FALSE;
   STATUS[285].EXT.BIT20 := FALSE;
   STATUS[285].EXT.AlarmSuppressed := FALSE;
   STATUS[285].EXT.AlarmPrsent := FALSE;
   STATUS[285].EXT.AlarmFailUnAck := FALSE;
   STATUS[285].Status := 0;
   STATUS[285].TimeStamp := 16#0000;
   STATUS[286].VALUE := 0.0;
   STATUS[286].TRIGVALUE := 0.0;
   STATUS[286].EXT.AlarmWarnUnAck := FALSE;
   STATUS[286].EXT.AckRequired := FALSE;
   STATUS[286].EXT.Maintanence := FALSE;
   STATUS[286].EXT.Operation := FALSE;
   STATUS[286].EXT.Forced := FALSE;
   STATUS[286].EXT.BIT29 := FALSE;
   STATUS[286].EXT.BIT30 := FALSE;
   STATUS[286].EXT.BIT31 := FALSE;
   STATUS[286].EXT.ModeBit1 := FALSE;
   STATUS[286].EXT.ModeBit2 := FALSE;
   STATUS[286].EXT.ModeBit3 := FALSE;
   STATUS[286].EXT.BIT19 := FALSE;
   STATUS[286].EXT.BIT20 := FALSE;
   STATUS[286].EXT.AlarmSuppressed := FALSE;
   STATUS[286].EXT.AlarmPrsent := FALSE;
   STATUS[286].EXT.AlarmFailUnAck := FALSE;
   STATUS[286].Status := 0;
   STATUS[286].TimeStamp := 16#0000;
   STATUS[287].VALUE := 0.0;
   STATUS[287].TRIGVALUE := 0.0;
   STATUS[287].EXT.AlarmWarnUnAck := FALSE;
   STATUS[287].EXT.AckRequired := FALSE;
   STATUS[287].EXT.Maintanence := FALSE;
   STATUS[287].EXT.Operation := FALSE;
   STATUS[287].EXT.Forced := FALSE;
   STATUS[287].EXT.BIT29 := FALSE;
   STATUS[287].EXT.BIT30 := FALSE;
   STATUS[287].EXT.BIT31 := FALSE;
   STATUS[287].EXT.ModeBit1 := FALSE;
   STATUS[287].EXT.ModeBit2 := FALSE;
   STATUS[287].EXT.ModeBit3 := FALSE;
   STATUS[287].EXT.BIT19 := FALSE;
   STATUS[287].EXT.BIT20 := FALSE;
   STATUS[287].EXT.AlarmSuppressed := FALSE;
   STATUS[287].EXT.AlarmPrsent := FALSE;
   STATUS[287].EXT.AlarmFailUnAck := FALSE;
   STATUS[287].Status := 0;
   STATUS[287].TimeStamp := 16#0000;
   STATUS[288].VALUE := 0.0;
   STATUS[288].TRIGVALUE := 0.0;
   STATUS[288].EXT.AlarmWarnUnAck := FALSE;
   STATUS[288].EXT.AckRequired := FALSE;
   STATUS[288].EXT.Maintanence := FALSE;
   STATUS[288].EXT.Operation := FALSE;
   STATUS[288].EXT.Forced := FALSE;
   STATUS[288].EXT.BIT29 := FALSE;
   STATUS[288].EXT.BIT30 := FALSE;
   STATUS[288].EXT.BIT31 := FALSE;
   STATUS[288].EXT.ModeBit1 := FALSE;
   STATUS[288].EXT.ModeBit2 := FALSE;
   STATUS[288].EXT.ModeBit3 := FALSE;
   STATUS[288].EXT.BIT19 := FALSE;
   STATUS[288].EXT.BIT20 := FALSE;
   STATUS[288].EXT.AlarmSuppressed := FALSE;
   STATUS[288].EXT.AlarmPrsent := FALSE;
   STATUS[288].EXT.AlarmFailUnAck := FALSE;
   STATUS[288].Status := 0;
   STATUS[288].TimeStamp := 16#0000;
   STATUS[289].VALUE := 0.0;
   STATUS[289].TRIGVALUE := 0.0;
   STATUS[289].EXT.AlarmWarnUnAck := FALSE;
   STATUS[289].EXT.AckRequired := FALSE;
   STATUS[289].EXT.Maintanence := FALSE;
   STATUS[289].EXT.Operation := FALSE;
   STATUS[289].EXT.Forced := FALSE;
   STATUS[289].EXT.BIT29 := FALSE;
   STATUS[289].EXT.BIT30 := FALSE;
   STATUS[289].EXT.BIT31 := FALSE;
   STATUS[289].EXT.ModeBit1 := FALSE;
   STATUS[289].EXT.ModeBit2 := FALSE;
   STATUS[289].EXT.ModeBit3 := FALSE;
   STATUS[289].EXT.BIT19 := FALSE;
   STATUS[289].EXT.BIT20 := FALSE;
   STATUS[289].EXT.AlarmSuppressed := FALSE;
   STATUS[289].EXT.AlarmPrsent := FALSE;
   STATUS[289].EXT.AlarmFailUnAck := FALSE;
   STATUS[289].Status := 0;
   STATUS[289].TimeStamp := 16#0000;
   STATUS[290].VALUE := 0.0;
   STATUS[290].TRIGVALUE := 0.0;
   STATUS[290].EXT.AlarmWarnUnAck := FALSE;
   STATUS[290].EXT.AckRequired := FALSE;
   STATUS[290].EXT.Maintanence := FALSE;
   STATUS[290].EXT.Operation := FALSE;
   STATUS[290].EXT.Forced := FALSE;
   STATUS[290].EXT.BIT29 := FALSE;
   STATUS[290].EXT.BIT30 := FALSE;
   STATUS[290].EXT.BIT31 := FALSE;
   STATUS[290].EXT.ModeBit1 := FALSE;
   STATUS[290].EXT.ModeBit2 := FALSE;
   STATUS[290].EXT.ModeBit3 := FALSE;
   STATUS[290].EXT.BIT19 := FALSE;
   STATUS[290].EXT.BIT20 := FALSE;
   STATUS[290].EXT.AlarmSuppressed := FALSE;
   STATUS[290].EXT.AlarmPrsent := FALSE;
   STATUS[290].EXT.AlarmFailUnAck := FALSE;
   STATUS[290].Status := 0;
   STATUS[290].TimeStamp := 16#0000;
   STATUS[291].VALUE := 0.0;
   STATUS[291].TRIGVALUE := 0.0;
   STATUS[291].EXT.AlarmWarnUnAck := FALSE;
   STATUS[291].EXT.AckRequired := FALSE;
   STATUS[291].EXT.Maintanence := FALSE;
   STATUS[291].EXT.Operation := FALSE;
   STATUS[291].EXT.Forced := FALSE;
   STATUS[291].EXT.BIT29 := FALSE;
   STATUS[291].EXT.BIT30 := FALSE;
   STATUS[291].EXT.BIT31 := FALSE;
   STATUS[291].EXT.ModeBit1 := FALSE;
   STATUS[291].EXT.ModeBit2 := FALSE;
   STATUS[291].EXT.ModeBit3 := FALSE;
   STATUS[291].EXT.BIT19 := FALSE;
   STATUS[291].EXT.BIT20 := FALSE;
   STATUS[291].EXT.AlarmSuppressed := FALSE;
   STATUS[291].EXT.AlarmPrsent := FALSE;
   STATUS[291].EXT.AlarmFailUnAck := FALSE;
   STATUS[291].Status := 0;
   STATUS[291].TimeStamp := 16#0000;
   STATUS[292].VALUE := 0.0;
   STATUS[292].TRIGVALUE := 0.0;
   STATUS[292].EXT.AlarmWarnUnAck := FALSE;
   STATUS[292].EXT.AckRequired := FALSE;
   STATUS[292].EXT.Maintanence := FALSE;
   STATUS[292].EXT.Operation := FALSE;
   STATUS[292].EXT.Forced := FALSE;
   STATUS[292].EXT.BIT29 := FALSE;
   STATUS[292].EXT.BIT30 := FALSE;
   STATUS[292].EXT.BIT31 := FALSE;
   STATUS[292].EXT.ModeBit1 := FALSE;
   STATUS[292].EXT.ModeBit2 := FALSE;
   STATUS[292].EXT.ModeBit3 := FALSE;
   STATUS[292].EXT.BIT19 := FALSE;
   STATUS[292].EXT.BIT20 := FALSE;
   STATUS[292].EXT.AlarmSuppressed := FALSE;
   STATUS[292].EXT.AlarmPrsent := FALSE;
   STATUS[292].EXT.AlarmFailUnAck := FALSE;
   STATUS[292].Status := 0;
   STATUS[292].TimeStamp := 16#0000;
   STATUS[293].VALUE := 0.0;
   STATUS[293].TRIGVALUE := 0.0;
   STATUS[293].EXT.AlarmWarnUnAck := FALSE;
   STATUS[293].EXT.AckRequired := FALSE;
   STATUS[293].EXT.Maintanence := FALSE;
   STATUS[293].EXT.Operation := FALSE;
   STATUS[293].EXT.Forced := FALSE;
   STATUS[293].EXT.BIT29 := FALSE;
   STATUS[293].EXT.BIT30 := FALSE;
   STATUS[293].EXT.BIT31 := FALSE;
   STATUS[293].EXT.ModeBit1 := FALSE;
   STATUS[293].EXT.ModeBit2 := FALSE;
   STATUS[293].EXT.ModeBit3 := FALSE;
   STATUS[293].EXT.BIT19 := FALSE;
   STATUS[293].EXT.BIT20 := FALSE;
   STATUS[293].EXT.AlarmSuppressed := FALSE;
   STATUS[293].EXT.AlarmPrsent := FALSE;
   STATUS[293].EXT.AlarmFailUnAck := FALSE;
   STATUS[293].Status := 0;
   STATUS[293].TimeStamp := 16#0000;
   STATUS[294].VALUE := 0.0;
   STATUS[294].TRIGVALUE := 0.0;
   STATUS[294].EXT.AlarmWarnUnAck := FALSE;
   STATUS[294].EXT.AckRequired := FALSE;
   STATUS[294].EXT.Maintanence := FALSE;
   STATUS[294].EXT.Operation := FALSE;
   STATUS[294].EXT.Forced := FALSE;
   STATUS[294].EXT.BIT29 := FALSE;
   STATUS[294].EXT.BIT30 := FALSE;
   STATUS[294].EXT.BIT31 := FALSE;
   STATUS[294].EXT.ModeBit1 := FALSE;
   STATUS[294].EXT.ModeBit2 := FALSE;
   STATUS[294].EXT.ModeBit3 := FALSE;
   STATUS[294].EXT.BIT19 := FALSE;
   STATUS[294].EXT.BIT20 := FALSE;
   STATUS[294].EXT.AlarmSuppressed := FALSE;
   STATUS[294].EXT.AlarmPrsent := FALSE;
   STATUS[294].EXT.AlarmFailUnAck := FALSE;
   STATUS[294].Status := 0;
   STATUS[294].TimeStamp := 16#0000;
   STATUS[295].VALUE := 0.0;
   STATUS[295].TRIGVALUE := 0.0;
   STATUS[295].EXT.AlarmWarnUnAck := FALSE;
   STATUS[295].EXT.AckRequired := FALSE;
   STATUS[295].EXT.Maintanence := FALSE;
   STATUS[295].EXT.Operation := FALSE;
   STATUS[295].EXT.Forced := FALSE;
   STATUS[295].EXT.BIT29 := FALSE;
   STATUS[295].EXT.BIT30 := FALSE;
   STATUS[295].EXT.BIT31 := FALSE;
   STATUS[295].EXT.ModeBit1 := FALSE;
   STATUS[295].EXT.ModeBit2 := FALSE;
   STATUS[295].EXT.ModeBit3 := FALSE;
   STATUS[295].EXT.BIT19 := FALSE;
   STATUS[295].EXT.BIT20 := FALSE;
   STATUS[295].EXT.AlarmSuppressed := FALSE;
   STATUS[295].EXT.AlarmPrsent := FALSE;
   STATUS[295].EXT.AlarmFailUnAck := FALSE;
   STATUS[295].Status := 0;
   STATUS[295].TimeStamp := 16#0000;
   STATUS[296].VALUE := 0.0;
   STATUS[296].TRIGVALUE := 0.0;
   STATUS[296].EXT.AlarmWarnUnAck := FALSE;
   STATUS[296].EXT.AckRequired := FALSE;
   STATUS[296].EXT.Maintanence := FALSE;
   STATUS[296].EXT.Operation := FALSE;
   STATUS[296].EXT.Forced := FALSE;
   STATUS[296].EXT.BIT29 := FALSE;
   STATUS[296].EXT.BIT30 := FALSE;
   STATUS[296].EXT.BIT31 := FALSE;
   STATUS[296].EXT.ModeBit1 := FALSE;
   STATUS[296].EXT.ModeBit2 := FALSE;
   STATUS[296].EXT.ModeBit3 := FALSE;
   STATUS[296].EXT.BIT19 := FALSE;
   STATUS[296].EXT.BIT20 := FALSE;
   STATUS[296].EXT.AlarmSuppressed := FALSE;
   STATUS[296].EXT.AlarmPrsent := FALSE;
   STATUS[296].EXT.AlarmFailUnAck := FALSE;
   STATUS[296].Status := 0;
   STATUS[296].TimeStamp := 16#0000;
   STATUS[297].VALUE := 0.0;
   STATUS[297].TRIGVALUE := 0.0;
   STATUS[297].EXT.AlarmWarnUnAck := FALSE;
   STATUS[297].EXT.AckRequired := FALSE;
   STATUS[297].EXT.Maintanence := FALSE;
   STATUS[297].EXT.Operation := FALSE;
   STATUS[297].EXT.Forced := FALSE;
   STATUS[297].EXT.BIT29 := FALSE;
   STATUS[297].EXT.BIT30 := FALSE;
   STATUS[297].EXT.BIT31 := FALSE;
   STATUS[297].EXT.ModeBit1 := FALSE;
   STATUS[297].EXT.ModeBit2 := FALSE;
   STATUS[297].EXT.ModeBit3 := FALSE;
   STATUS[297].EXT.BIT19 := FALSE;
   STATUS[297].EXT.BIT20 := FALSE;
   STATUS[297].EXT.AlarmSuppressed := FALSE;
   STATUS[297].EXT.AlarmPrsent := FALSE;
   STATUS[297].EXT.AlarmFailUnAck := FALSE;
   STATUS[297].Status := 0;
   STATUS[297].TimeStamp := 16#0000;
   STATUS[298].VALUE := 0.0;
   STATUS[298].TRIGVALUE := 0.0;
   STATUS[298].EXT.AlarmWarnUnAck := FALSE;
   STATUS[298].EXT.AckRequired := FALSE;
   STATUS[298].EXT.Maintanence := FALSE;
   STATUS[298].EXT.Operation := FALSE;
   STATUS[298].EXT.Forced := FALSE;
   STATUS[298].EXT.BIT29 := FALSE;
   STATUS[298].EXT.BIT30 := FALSE;
   STATUS[298].EXT.BIT31 := FALSE;
   STATUS[298].EXT.ModeBit1 := FALSE;
   STATUS[298].EXT.ModeBit2 := FALSE;
   STATUS[298].EXT.ModeBit3 := FALSE;
   STATUS[298].EXT.BIT19 := FALSE;
   STATUS[298].EXT.BIT20 := FALSE;
   STATUS[298].EXT.AlarmSuppressed := FALSE;
   STATUS[298].EXT.AlarmPrsent := FALSE;
   STATUS[298].EXT.AlarmFailUnAck := FALSE;
   STATUS[298].Status := 0;
   STATUS[298].TimeStamp := 16#0000;
   STATUS[299].VALUE := 0.0;
   STATUS[299].TRIGVALUE := 0.0;
   STATUS[299].EXT.AlarmWarnUnAck := FALSE;
   STATUS[299].EXT.AckRequired := FALSE;
   STATUS[299].EXT.Maintanence := FALSE;
   STATUS[299].EXT.Operation := FALSE;
   STATUS[299].EXT.Forced := FALSE;
   STATUS[299].EXT.BIT29 := FALSE;
   STATUS[299].EXT.BIT30 := FALSE;
   STATUS[299].EXT.BIT31 := FALSE;
   STATUS[299].EXT.ModeBit1 := FALSE;
   STATUS[299].EXT.ModeBit2 := FALSE;
   STATUS[299].EXT.ModeBit3 := FALSE;
   STATUS[299].EXT.BIT19 := FALSE;
   STATUS[299].EXT.BIT20 := FALSE;
   STATUS[299].EXT.AlarmSuppressed := FALSE;
   STATUS[299].EXT.AlarmPrsent := FALSE;
   STATUS[299].EXT.AlarmFailUnAck := FALSE;
   STATUS[299].Status := 0;
   STATUS[299].TimeStamp := 16#0000;
   STATUS[300].VALUE := 0.0;
   STATUS[300].TRIGVALUE := 0.0;
   STATUS[300].EXT.AlarmWarnUnAck := FALSE;
   STATUS[300].EXT.AckRequired := FALSE;
   STATUS[300].EXT.Maintanence := FALSE;
   STATUS[300].EXT.Operation := FALSE;
   STATUS[300].EXT.Forced := FALSE;
   STATUS[300].EXT.BIT29 := FALSE;
   STATUS[300].EXT.BIT30 := FALSE;
   STATUS[300].EXT.BIT31 := FALSE;
   STATUS[300].EXT.ModeBit1 := FALSE;
   STATUS[300].EXT.ModeBit2 := FALSE;
   STATUS[300].EXT.ModeBit3 := FALSE;
   STATUS[300].EXT.BIT19 := FALSE;
   STATUS[300].EXT.BIT20 := FALSE;
   STATUS[300].EXT.AlarmSuppressed := FALSE;
   STATUS[300].EXT.AlarmPrsent := FALSE;
   STATUS[300].EXT.AlarmFailUnAck := FALSE;
   STATUS[300].Status := 0;
   STATUS[300].TimeStamp := 16#0000;
   STATUS[301].VALUE := 0.0;
   STATUS[301].TRIGVALUE := 0.0;
   STATUS[301].EXT.AlarmWarnUnAck := FALSE;
   STATUS[301].EXT.AckRequired := FALSE;
   STATUS[301].EXT.Maintanence := FALSE;
   STATUS[301].EXT.Operation := FALSE;
   STATUS[301].EXT.Forced := FALSE;
   STATUS[301].EXT.BIT29 := FALSE;
   STATUS[301].EXT.BIT30 := FALSE;
   STATUS[301].EXT.BIT31 := FALSE;
   STATUS[301].EXT.ModeBit1 := FALSE;
   STATUS[301].EXT.ModeBit2 := FALSE;
   STATUS[301].EXT.ModeBit3 := FALSE;
   STATUS[301].EXT.BIT19 := FALSE;
   STATUS[301].EXT.BIT20 := FALSE;
   STATUS[301].EXT.AlarmSuppressed := FALSE;
   STATUS[301].EXT.AlarmPrsent := FALSE;
   STATUS[301].EXT.AlarmFailUnAck := FALSE;
   STATUS[301].Status := 0;
   STATUS[301].TimeStamp := 16#0000;
   STATUS[302].VALUE := 0.0;
   STATUS[302].TRIGVALUE := 0.0;
   STATUS[302].EXT.AlarmWarnUnAck := FALSE;
   STATUS[302].EXT.AckRequired := FALSE;
   STATUS[302].EXT.Maintanence := FALSE;
   STATUS[302].EXT.Operation := FALSE;
   STATUS[302].EXT.Forced := FALSE;
   STATUS[302].EXT.BIT29 := FALSE;
   STATUS[302].EXT.BIT30 := FALSE;
   STATUS[302].EXT.BIT31 := FALSE;
   STATUS[302].EXT.ModeBit1 := FALSE;
   STATUS[302].EXT.ModeBit2 := FALSE;
   STATUS[302].EXT.ModeBit3 := FALSE;
   STATUS[302].EXT.BIT19 := FALSE;
   STATUS[302].EXT.BIT20 := FALSE;
   STATUS[302].EXT.AlarmSuppressed := FALSE;
   STATUS[302].EXT.AlarmPrsent := FALSE;
   STATUS[302].EXT.AlarmFailUnAck := FALSE;
   STATUS[302].Status := 0;
   STATUS[302].TimeStamp := 16#0000;
   STATUS[303].VALUE := 0.0;
   STATUS[303].TRIGVALUE := 0.0;
   STATUS[303].EXT.AlarmWarnUnAck := FALSE;
   STATUS[303].EXT.AckRequired := FALSE;
   STATUS[303].EXT.Maintanence := FALSE;
   STATUS[303].EXT.Operation := FALSE;
   STATUS[303].EXT.Forced := FALSE;
   STATUS[303].EXT.BIT29 := FALSE;
   STATUS[303].EXT.BIT30 := FALSE;
   STATUS[303].EXT.BIT31 := FALSE;
   STATUS[303].EXT.ModeBit1 := FALSE;
   STATUS[303].EXT.ModeBit2 := FALSE;
   STATUS[303].EXT.ModeBit3 := FALSE;
   STATUS[303].EXT.BIT19 := FALSE;
   STATUS[303].EXT.BIT20 := FALSE;
   STATUS[303].EXT.AlarmSuppressed := FALSE;
   STATUS[303].EXT.AlarmPrsent := FALSE;
   STATUS[303].EXT.AlarmFailUnAck := FALSE;
   STATUS[303].Status := 0;
   STATUS[303].TimeStamp := 16#0000;
   STATUS[304].VALUE := 0.0;
   STATUS[304].TRIGVALUE := 0.0;
   STATUS[304].EXT.AlarmWarnUnAck := FALSE;
   STATUS[304].EXT.AckRequired := FALSE;
   STATUS[304].EXT.Maintanence := FALSE;
   STATUS[304].EXT.Operation := FALSE;
   STATUS[304].EXT.Forced := FALSE;
   STATUS[304].EXT.BIT29 := FALSE;
   STATUS[304].EXT.BIT30 := FALSE;
   STATUS[304].EXT.BIT31 := FALSE;
   STATUS[304].EXT.ModeBit1 := FALSE;
   STATUS[304].EXT.ModeBit2 := FALSE;
   STATUS[304].EXT.ModeBit3 := FALSE;
   STATUS[304].EXT.BIT19 := FALSE;
   STATUS[304].EXT.BIT20 := FALSE;
   STATUS[304].EXT.AlarmSuppressed := FALSE;
   STATUS[304].EXT.AlarmPrsent := FALSE;
   STATUS[304].EXT.AlarmFailUnAck := FALSE;
   STATUS[304].Status := 0;
   STATUS[304].TimeStamp := 16#0000;
   STATUS[305].VALUE := 0.0;
   STATUS[305].TRIGVALUE := 0.0;
   STATUS[305].EXT.AlarmWarnUnAck := FALSE;
   STATUS[305].EXT.AckRequired := FALSE;
   STATUS[305].EXT.Maintanence := FALSE;
   STATUS[305].EXT.Operation := FALSE;
   STATUS[305].EXT.Forced := FALSE;
   STATUS[305].EXT.BIT29 := FALSE;
   STATUS[305].EXT.BIT30 := FALSE;
   STATUS[305].EXT.BIT31 := FALSE;
   STATUS[305].EXT.ModeBit1 := FALSE;
   STATUS[305].EXT.ModeBit2 := FALSE;
   STATUS[305].EXT.ModeBit3 := FALSE;
   STATUS[305].EXT.BIT19 := FALSE;
   STATUS[305].EXT.BIT20 := FALSE;
   STATUS[305].EXT.AlarmSuppressed := FALSE;
   STATUS[305].EXT.AlarmPrsent := FALSE;
   STATUS[305].EXT.AlarmFailUnAck := FALSE;
   STATUS[305].Status := 0;
   STATUS[305].TimeStamp := 16#0000;
   STATUS[306].VALUE := 0.0;
   STATUS[306].TRIGVALUE := 0.0;
   STATUS[306].EXT.AlarmWarnUnAck := FALSE;
   STATUS[306].EXT.AckRequired := FALSE;
   STATUS[306].EXT.Maintanence := FALSE;
   STATUS[306].EXT.Operation := FALSE;
   STATUS[306].EXT.Forced := FALSE;
   STATUS[306].EXT.BIT29 := FALSE;
   STATUS[306].EXT.BIT30 := FALSE;
   STATUS[306].EXT.BIT31 := FALSE;
   STATUS[306].EXT.ModeBit1 := FALSE;
   STATUS[306].EXT.ModeBit2 := FALSE;
   STATUS[306].EXT.ModeBit3 := FALSE;
   STATUS[306].EXT.BIT19 := FALSE;
   STATUS[306].EXT.BIT20 := FALSE;
   STATUS[306].EXT.AlarmSuppressed := FALSE;
   STATUS[306].EXT.AlarmPrsent := FALSE;
   STATUS[306].EXT.AlarmFailUnAck := FALSE;
   STATUS[306].Status := 0;
   STATUS[306].TimeStamp := 16#0000;
   STATUS[307].VALUE := 0.0;
   STATUS[307].TRIGVALUE := 0.0;
   STATUS[307].EXT.AlarmWarnUnAck := FALSE;
   STATUS[307].EXT.AckRequired := FALSE;
   STATUS[307].EXT.Maintanence := FALSE;
   STATUS[307].EXT.Operation := FALSE;
   STATUS[307].EXT.Forced := FALSE;
   STATUS[307].EXT.BIT29 := FALSE;
   STATUS[307].EXT.BIT30 := FALSE;
   STATUS[307].EXT.BIT31 := FALSE;
   STATUS[307].EXT.ModeBit1 := FALSE;
   STATUS[307].EXT.ModeBit2 := FALSE;
   STATUS[307].EXT.ModeBit3 := FALSE;
   STATUS[307].EXT.BIT19 := FALSE;
   STATUS[307].EXT.BIT20 := FALSE;
   STATUS[307].EXT.AlarmSuppressed := FALSE;
   STATUS[307].EXT.AlarmPrsent := FALSE;
   STATUS[307].EXT.AlarmFailUnAck := FALSE;
   STATUS[307].Status := 0;
   STATUS[307].TimeStamp := 16#0000;
   STATUS[308].VALUE := 0.0;
   STATUS[308].TRIGVALUE := 0.0;
   STATUS[308].EXT.AlarmWarnUnAck := FALSE;
   STATUS[308].EXT.AckRequired := FALSE;
   STATUS[308].EXT.Maintanence := FALSE;
   STATUS[308].EXT.Operation := FALSE;
   STATUS[308].EXT.Forced := FALSE;
   STATUS[308].EXT.BIT29 := FALSE;
   STATUS[308].EXT.BIT30 := FALSE;
   STATUS[308].EXT.BIT31 := FALSE;
   STATUS[308].EXT.ModeBit1 := FALSE;
   STATUS[308].EXT.ModeBit2 := FALSE;
   STATUS[308].EXT.ModeBit3 := FALSE;
   STATUS[308].EXT.BIT19 := FALSE;
   STATUS[308].EXT.BIT20 := FALSE;
   STATUS[308].EXT.AlarmSuppressed := FALSE;
   STATUS[308].EXT.AlarmPrsent := FALSE;
   STATUS[308].EXT.AlarmFailUnAck := FALSE;
   STATUS[308].Status := 0;
   STATUS[308].TimeStamp := 16#0000;
   STATUS[309].VALUE := 0.0;
   STATUS[309].TRIGVALUE := 0.0;
   STATUS[309].EXT.AlarmWarnUnAck := FALSE;
   STATUS[309].EXT.AckRequired := FALSE;
   STATUS[309].EXT.Maintanence := FALSE;
   STATUS[309].EXT.Operation := FALSE;
   STATUS[309].EXT.Forced := FALSE;
   STATUS[309].EXT.BIT29 := FALSE;
   STATUS[309].EXT.BIT30 := FALSE;
   STATUS[309].EXT.BIT31 := FALSE;
   STATUS[309].EXT.ModeBit1 := FALSE;
   STATUS[309].EXT.ModeBit2 := FALSE;
   STATUS[309].EXT.ModeBit3 := FALSE;
   STATUS[309].EXT.BIT19 := FALSE;
   STATUS[309].EXT.BIT20 := FALSE;
   STATUS[309].EXT.AlarmSuppressed := FALSE;
   STATUS[309].EXT.AlarmPrsent := FALSE;
   STATUS[309].EXT.AlarmFailUnAck := FALSE;
   STATUS[309].Status := 0;
   STATUS[309].TimeStamp := 16#0000;
   STATUS[310].VALUE := 0.0;
   STATUS[310].TRIGVALUE := 0.0;
   STATUS[310].EXT.AlarmWarnUnAck := FALSE;
   STATUS[310].EXT.AckRequired := FALSE;
   STATUS[310].EXT.Maintanence := FALSE;
   STATUS[310].EXT.Operation := FALSE;
   STATUS[310].EXT.Forced := FALSE;
   STATUS[310].EXT.BIT29 := FALSE;
   STATUS[310].EXT.BIT30 := FALSE;
   STATUS[310].EXT.BIT31 := FALSE;
   STATUS[310].EXT.ModeBit1 := FALSE;
   STATUS[310].EXT.ModeBit2 := FALSE;
   STATUS[310].EXT.ModeBit3 := FALSE;
   STATUS[310].EXT.BIT19 := FALSE;
   STATUS[310].EXT.BIT20 := FALSE;
   STATUS[310].EXT.AlarmSuppressed := FALSE;
   STATUS[310].EXT.AlarmPrsent := FALSE;
   STATUS[310].EXT.AlarmFailUnAck := FALSE;
   STATUS[310].Status := 0;
   STATUS[310].TimeStamp := 16#0000;
   STATUS[311].VALUE := 0.0;
   STATUS[311].TRIGVALUE := 0.0;
   STATUS[311].EXT.AlarmWarnUnAck := FALSE;
   STATUS[311].EXT.AckRequired := FALSE;
   STATUS[311].EXT.Maintanence := FALSE;
   STATUS[311].EXT.Operation := FALSE;
   STATUS[311].EXT.Forced := FALSE;
   STATUS[311].EXT.BIT29 := FALSE;
   STATUS[311].EXT.BIT30 := FALSE;
   STATUS[311].EXT.BIT31 := FALSE;
   STATUS[311].EXT.ModeBit1 := FALSE;
   STATUS[311].EXT.ModeBit2 := FALSE;
   STATUS[311].EXT.ModeBit3 := FALSE;
   STATUS[311].EXT.BIT19 := FALSE;
   STATUS[311].EXT.BIT20 := FALSE;
   STATUS[311].EXT.AlarmSuppressed := FALSE;
   STATUS[311].EXT.AlarmPrsent := FALSE;
   STATUS[311].EXT.AlarmFailUnAck := FALSE;
   STATUS[311].Status := 0;
   STATUS[311].TimeStamp := 16#0000;
   STATUS[312].VALUE := 0.0;
   STATUS[312].TRIGVALUE := 0.0;
   STATUS[312].EXT.AlarmWarnUnAck := FALSE;
   STATUS[312].EXT.AckRequired := FALSE;
   STATUS[312].EXT.Maintanence := FALSE;
   STATUS[312].EXT.Operation := FALSE;
   STATUS[312].EXT.Forced := FALSE;
   STATUS[312].EXT.BIT29 := FALSE;
   STATUS[312].EXT.BIT30 := FALSE;
   STATUS[312].EXT.BIT31 := FALSE;
   STATUS[312].EXT.ModeBit1 := FALSE;
   STATUS[312].EXT.ModeBit2 := FALSE;
   STATUS[312].EXT.ModeBit3 := FALSE;
   STATUS[312].EXT.BIT19 := FALSE;
   STATUS[312].EXT.BIT20 := FALSE;
   STATUS[312].EXT.AlarmSuppressed := FALSE;
   STATUS[312].EXT.AlarmPrsent := FALSE;
   STATUS[312].EXT.AlarmFailUnAck := FALSE;
   STATUS[312].Status := 0;
   STATUS[312].TimeStamp := 16#0000;
   STATUS[313].VALUE := 0.0;
   STATUS[313].TRIGVALUE := 0.0;
   STATUS[313].EXT.AlarmWarnUnAck := FALSE;
   STATUS[313].EXT.AckRequired := FALSE;
   STATUS[313].EXT.Maintanence := FALSE;
   STATUS[313].EXT.Operation := FALSE;
   STATUS[313].EXT.Forced := FALSE;
   STATUS[313].EXT.BIT29 := FALSE;
   STATUS[313].EXT.BIT30 := FALSE;
   STATUS[313].EXT.BIT31 := FALSE;
   STATUS[313].EXT.ModeBit1 := FALSE;
   STATUS[313].EXT.ModeBit2 := FALSE;
   STATUS[313].EXT.ModeBit3 := FALSE;
   STATUS[313].EXT.BIT19 := FALSE;
   STATUS[313].EXT.BIT20 := FALSE;
   STATUS[313].EXT.AlarmSuppressed := FALSE;
   STATUS[313].EXT.AlarmPrsent := FALSE;
   STATUS[313].EXT.AlarmFailUnAck := FALSE;
   STATUS[313].Status := 0;
   STATUS[313].TimeStamp := 16#0000;
   STATUS[314].VALUE := 0.0;
   STATUS[314].TRIGVALUE := 0.0;
   STATUS[314].EXT.AlarmWarnUnAck := FALSE;
   STATUS[314].EXT.AckRequired := FALSE;
   STATUS[314].EXT.Maintanence := FALSE;
   STATUS[314].EXT.Operation := FALSE;
   STATUS[314].EXT.Forced := FALSE;
   STATUS[314].EXT.BIT29 := FALSE;
   STATUS[314].EXT.BIT30 := FALSE;
   STATUS[314].EXT.BIT31 := FALSE;
   STATUS[314].EXT.ModeBit1 := FALSE;
   STATUS[314].EXT.ModeBit2 := FALSE;
   STATUS[314].EXT.ModeBit3 := FALSE;
   STATUS[314].EXT.BIT19 := FALSE;
   STATUS[314].EXT.BIT20 := FALSE;
   STATUS[314].EXT.AlarmSuppressed := FALSE;
   STATUS[314].EXT.AlarmPrsent := FALSE;
   STATUS[314].EXT.AlarmFailUnAck := FALSE;
   STATUS[314].Status := 0;
   STATUS[314].TimeStamp := 16#0000;
   STATUS[315].VALUE := 0.0;
   STATUS[315].TRIGVALUE := 0.0;
   STATUS[315].EXT.AlarmWarnUnAck := FALSE;
   STATUS[315].EXT.AckRequired := FALSE;
   STATUS[315].EXT.Maintanence := FALSE;
   STATUS[315].EXT.Operation := FALSE;
   STATUS[315].EXT.Forced := FALSE;
   STATUS[315].EXT.BIT29 := FALSE;
   STATUS[315].EXT.BIT30 := FALSE;
   STATUS[315].EXT.BIT31 := FALSE;
   STATUS[315].EXT.ModeBit1 := FALSE;
   STATUS[315].EXT.ModeBit2 := FALSE;
   STATUS[315].EXT.ModeBit3 := FALSE;
   STATUS[315].EXT.BIT19 := FALSE;
   STATUS[315].EXT.BIT20 := FALSE;
   STATUS[315].EXT.AlarmSuppressed := FALSE;
   STATUS[315].EXT.AlarmPrsent := FALSE;
   STATUS[315].EXT.AlarmFailUnAck := FALSE;
   STATUS[315].Status := 0;
   STATUS[315].TimeStamp := 16#0000;
   STATUS[316].VALUE := 0.0;
   STATUS[316].TRIGVALUE := 0.0;
   STATUS[316].EXT.AlarmWarnUnAck := FALSE;
   STATUS[316].EXT.AckRequired := FALSE;
   STATUS[316].EXT.Maintanence := FALSE;
   STATUS[316].EXT.Operation := FALSE;
   STATUS[316].EXT.Forced := FALSE;
   STATUS[316].EXT.BIT29 := FALSE;
   STATUS[316].EXT.BIT30 := FALSE;
   STATUS[316].EXT.BIT31 := FALSE;
   STATUS[316].EXT.ModeBit1 := FALSE;
   STATUS[316].EXT.ModeBit2 := FALSE;
   STATUS[316].EXT.ModeBit3 := FALSE;
   STATUS[316].EXT.BIT19 := FALSE;
   STATUS[316].EXT.BIT20 := FALSE;
   STATUS[316].EXT.AlarmSuppressed := FALSE;
   STATUS[316].EXT.AlarmPrsent := FALSE;
   STATUS[316].EXT.AlarmFailUnAck := FALSE;
   STATUS[316].Status := 0;
   STATUS[316].TimeStamp := 16#0000;
   STATUS[317].VALUE := 0.0;
   STATUS[317].TRIGVALUE := 0.0;
   STATUS[317].EXT.AlarmWarnUnAck := FALSE;
   STATUS[317].EXT.AckRequired := FALSE;
   STATUS[317].EXT.Maintanence := FALSE;
   STATUS[317].EXT.Operation := FALSE;
   STATUS[317].EXT.Forced := FALSE;
   STATUS[317].EXT.BIT29 := FALSE;
   STATUS[317].EXT.BIT30 := FALSE;
   STATUS[317].EXT.BIT31 := FALSE;
   STATUS[317].EXT.ModeBit1 := FALSE;
   STATUS[317].EXT.ModeBit2 := FALSE;
   STATUS[317].EXT.ModeBit3 := FALSE;
   STATUS[317].EXT.BIT19 := FALSE;
   STATUS[317].EXT.BIT20 := FALSE;
   STATUS[317].EXT.AlarmSuppressed := FALSE;
   STATUS[317].EXT.AlarmPrsent := FALSE;
   STATUS[317].EXT.AlarmFailUnAck := FALSE;
   STATUS[317].Status := 0;
   STATUS[317].TimeStamp := 16#0000;
   STATUS[318].VALUE := 0.0;
   STATUS[318].TRIGVALUE := 0.0;
   STATUS[318].EXT.AlarmWarnUnAck := FALSE;
   STATUS[318].EXT.AckRequired := FALSE;
   STATUS[318].EXT.Maintanence := FALSE;
   STATUS[318].EXT.Operation := FALSE;
   STATUS[318].EXT.Forced := FALSE;
   STATUS[318].EXT.BIT29 := FALSE;
   STATUS[318].EXT.BIT30 := FALSE;
   STATUS[318].EXT.BIT31 := FALSE;
   STATUS[318].EXT.ModeBit1 := FALSE;
   STATUS[318].EXT.ModeBit2 := FALSE;
   STATUS[318].EXT.ModeBit3 := FALSE;
   STATUS[318].EXT.BIT19 := FALSE;
   STATUS[318].EXT.BIT20 := FALSE;
   STATUS[318].EXT.AlarmSuppressed := FALSE;
   STATUS[318].EXT.AlarmPrsent := FALSE;
   STATUS[318].EXT.AlarmFailUnAck := FALSE;
   STATUS[318].Status := 0;
   STATUS[318].TimeStamp := 16#0000;
   STATUS[319].VALUE := 0.0;
   STATUS[319].TRIGVALUE := 0.0;
   STATUS[319].EXT.AlarmWarnUnAck := FALSE;
   STATUS[319].EXT.AckRequired := FALSE;
   STATUS[319].EXT.Maintanence := FALSE;
   STATUS[319].EXT.Operation := FALSE;
   STATUS[319].EXT.Forced := FALSE;
   STATUS[319].EXT.BIT29 := FALSE;
   STATUS[319].EXT.BIT30 := FALSE;
   STATUS[319].EXT.BIT31 := FALSE;
   STATUS[319].EXT.ModeBit1 := FALSE;
   STATUS[319].EXT.ModeBit2 := FALSE;
   STATUS[319].EXT.ModeBit3 := FALSE;
   STATUS[319].EXT.BIT19 := FALSE;
   STATUS[319].EXT.BIT20 := FALSE;
   STATUS[319].EXT.AlarmSuppressed := FALSE;
   STATUS[319].EXT.AlarmPrsent := FALSE;
   STATUS[319].EXT.AlarmFailUnAck := FALSE;
   STATUS[319].Status := 0;
   STATUS[319].TimeStamp := 16#0000;
   STATUS[320].VALUE := 0.0;
   STATUS[320].TRIGVALUE := 0.0;
   STATUS[320].EXT.AlarmWarnUnAck := FALSE;
   STATUS[320].EXT.AckRequired := FALSE;
   STATUS[320].EXT.Maintanence := FALSE;
   STATUS[320].EXT.Operation := FALSE;
   STATUS[320].EXT.Forced := FALSE;
   STATUS[320].EXT.BIT29 := FALSE;
   STATUS[320].EXT.BIT30 := FALSE;
   STATUS[320].EXT.BIT31 := FALSE;
   STATUS[320].EXT.ModeBit1 := FALSE;
   STATUS[320].EXT.ModeBit2 := FALSE;
   STATUS[320].EXT.ModeBit3 := FALSE;
   STATUS[320].EXT.BIT19 := FALSE;
   STATUS[320].EXT.BIT20 := FALSE;
   STATUS[320].EXT.AlarmSuppressed := FALSE;
   STATUS[320].EXT.AlarmPrsent := FALSE;
   STATUS[320].EXT.AlarmFailUnAck := FALSE;
   STATUS[320].Status := 0;
   STATUS[320].TimeStamp := 16#0000;
   STATUS[321].VALUE := 0.0;
   STATUS[321].TRIGVALUE := 0.0;
   STATUS[321].EXT.AlarmWarnUnAck := FALSE;
   STATUS[321].EXT.AckRequired := FALSE;
   STATUS[321].EXT.Maintanence := FALSE;
   STATUS[321].EXT.Operation := FALSE;
   STATUS[321].EXT.Forced := FALSE;
   STATUS[321].EXT.BIT29 := FALSE;
   STATUS[321].EXT.BIT30 := FALSE;
   STATUS[321].EXT.BIT31 := FALSE;
   STATUS[321].EXT.ModeBit1 := FALSE;
   STATUS[321].EXT.ModeBit2 := FALSE;
   STATUS[321].EXT.ModeBit3 := FALSE;
   STATUS[321].EXT.BIT19 := FALSE;
   STATUS[321].EXT.BIT20 := FALSE;
   STATUS[321].EXT.AlarmSuppressed := FALSE;
   STATUS[321].EXT.AlarmPrsent := FALSE;
   STATUS[321].EXT.AlarmFailUnAck := FALSE;
   STATUS[321].Status := 0;
   STATUS[321].TimeStamp := 16#0000;
   STATUS[322].VALUE := 0.0;
   STATUS[322].TRIGVALUE := 0.0;
   STATUS[322].EXT.AlarmWarnUnAck := FALSE;
   STATUS[322].EXT.AckRequired := FALSE;
   STATUS[322].EXT.Maintanence := FALSE;
   STATUS[322].EXT.Operation := FALSE;
   STATUS[322].EXT.Forced := FALSE;
   STATUS[322].EXT.BIT29 := FALSE;
   STATUS[322].EXT.BIT30 := FALSE;
   STATUS[322].EXT.BIT31 := FALSE;
   STATUS[322].EXT.ModeBit1 := FALSE;
   STATUS[322].EXT.ModeBit2 := FALSE;
   STATUS[322].EXT.ModeBit3 := FALSE;
   STATUS[322].EXT.BIT19 := FALSE;
   STATUS[322].EXT.BIT20 := FALSE;
   STATUS[322].EXT.AlarmSuppressed := FALSE;
   STATUS[322].EXT.AlarmPrsent := FALSE;
   STATUS[322].EXT.AlarmFailUnAck := FALSE;
   STATUS[322].Status := 0;
   STATUS[322].TimeStamp := 16#0000;
   STATUS[323].VALUE := 0.0;
   STATUS[323].TRIGVALUE := 0.0;
   STATUS[323].EXT.AlarmWarnUnAck := FALSE;
   STATUS[323].EXT.AckRequired := FALSE;
   STATUS[323].EXT.Maintanence := FALSE;
   STATUS[323].EXT.Operation := FALSE;
   STATUS[323].EXT.Forced := FALSE;
   STATUS[323].EXT.BIT29 := FALSE;
   STATUS[323].EXT.BIT30 := FALSE;
   STATUS[323].EXT.BIT31 := FALSE;
   STATUS[323].EXT.ModeBit1 := FALSE;
   STATUS[323].EXT.ModeBit2 := FALSE;
   STATUS[323].EXT.ModeBit3 := FALSE;
   STATUS[323].EXT.BIT19 := FALSE;
   STATUS[323].EXT.BIT20 := FALSE;
   STATUS[323].EXT.AlarmSuppressed := FALSE;
   STATUS[323].EXT.AlarmPrsent := FALSE;
   STATUS[323].EXT.AlarmFailUnAck := FALSE;
   STATUS[323].Status := 0;
   STATUS[323].TimeStamp := 16#0000;
   STATUS[324].VALUE := 0.0;
   STATUS[324].TRIGVALUE := 0.0;
   STATUS[324].EXT.AlarmWarnUnAck := FALSE;
   STATUS[324].EXT.AckRequired := FALSE;
   STATUS[324].EXT.Maintanence := FALSE;
   STATUS[324].EXT.Operation := FALSE;
   STATUS[324].EXT.Forced := FALSE;
   STATUS[324].EXT.BIT29 := FALSE;
   STATUS[324].EXT.BIT30 := FALSE;
   STATUS[324].EXT.BIT31 := FALSE;
   STATUS[324].EXT.ModeBit1 := FALSE;
   STATUS[324].EXT.ModeBit2 := FALSE;
   STATUS[324].EXT.ModeBit3 := FALSE;
   STATUS[324].EXT.BIT19 := FALSE;
   STATUS[324].EXT.BIT20 := FALSE;
   STATUS[324].EXT.AlarmSuppressed := FALSE;
   STATUS[324].EXT.AlarmPrsent := FALSE;
   STATUS[324].EXT.AlarmFailUnAck := FALSE;
   STATUS[324].Status := 0;
   STATUS[324].TimeStamp := 16#0000;
   STATUS[325].VALUE := 0.0;
   STATUS[325].TRIGVALUE := 0.0;
   STATUS[325].EXT.AlarmWarnUnAck := FALSE;
   STATUS[325].EXT.AckRequired := FALSE;
   STATUS[325].EXT.Maintanence := FALSE;
   STATUS[325].EXT.Operation := FALSE;
   STATUS[325].EXT.Forced := FALSE;
   STATUS[325].EXT.BIT29 := FALSE;
   STATUS[325].EXT.BIT30 := FALSE;
   STATUS[325].EXT.BIT31 := FALSE;
   STATUS[325].EXT.ModeBit1 := FALSE;
   STATUS[325].EXT.ModeBit2 := FALSE;
   STATUS[325].EXT.ModeBit3 := FALSE;
   STATUS[325].EXT.BIT19 := FALSE;
   STATUS[325].EXT.BIT20 := FALSE;
   STATUS[325].EXT.AlarmSuppressed := FALSE;
   STATUS[325].EXT.AlarmPrsent := FALSE;
   STATUS[325].EXT.AlarmFailUnAck := FALSE;
   STATUS[325].Status := 0;
   STATUS[325].TimeStamp := 16#0000;
   STATUS[326].VALUE := 0.0;
   STATUS[326].TRIGVALUE := 0.0;
   STATUS[326].EXT.AlarmWarnUnAck := FALSE;
   STATUS[326].EXT.AckRequired := FALSE;
   STATUS[326].EXT.Maintanence := FALSE;
   STATUS[326].EXT.Operation := FALSE;
   STATUS[326].EXT.Forced := FALSE;
   STATUS[326].EXT.BIT29 := FALSE;
   STATUS[326].EXT.BIT30 := FALSE;
   STATUS[326].EXT.BIT31 := FALSE;
   STATUS[326].EXT.ModeBit1 := FALSE;
   STATUS[326].EXT.ModeBit2 := FALSE;
   STATUS[326].EXT.ModeBit3 := FALSE;
   STATUS[326].EXT.BIT19 := FALSE;
   STATUS[326].EXT.BIT20 := FALSE;
   STATUS[326].EXT.AlarmSuppressed := FALSE;
   STATUS[326].EXT.AlarmPrsent := FALSE;
   STATUS[326].EXT.AlarmFailUnAck := FALSE;
   STATUS[326].Status := 0;
   STATUS[326].TimeStamp := 16#0000;
   STATUS[327].VALUE := 0.0;
   STATUS[327].TRIGVALUE := 0.0;
   STATUS[327].EXT.AlarmWarnUnAck := FALSE;
   STATUS[327].EXT.AckRequired := FALSE;
   STATUS[327].EXT.Maintanence := FALSE;
   STATUS[327].EXT.Operation := FALSE;
   STATUS[327].EXT.Forced := FALSE;
   STATUS[327].EXT.BIT29 := FALSE;
   STATUS[327].EXT.BIT30 := FALSE;
   STATUS[327].EXT.BIT31 := FALSE;
   STATUS[327].EXT.ModeBit1 := FALSE;
   STATUS[327].EXT.ModeBit2 := FALSE;
   STATUS[327].EXT.ModeBit3 := FALSE;
   STATUS[327].EXT.BIT19 := FALSE;
   STATUS[327].EXT.BIT20 := FALSE;
   STATUS[327].EXT.AlarmSuppressed := FALSE;
   STATUS[327].EXT.AlarmPrsent := FALSE;
   STATUS[327].EXT.AlarmFailUnAck := FALSE;
   STATUS[327].Status := 0;
   STATUS[327].TimeStamp := 16#0000;
   STATUS[328].VALUE := 0.0;
   STATUS[328].TRIGVALUE := 0.0;
   STATUS[328].EXT.AlarmWarnUnAck := FALSE;
   STATUS[328].EXT.AckRequired := FALSE;
   STATUS[328].EXT.Maintanence := FALSE;
   STATUS[328].EXT.Operation := FALSE;
   STATUS[328].EXT.Forced := FALSE;
   STATUS[328].EXT.BIT29 := FALSE;
   STATUS[328].EXT.BIT30 := FALSE;
   STATUS[328].EXT.BIT31 := FALSE;
   STATUS[328].EXT.ModeBit1 := FALSE;
   STATUS[328].EXT.ModeBit2 := FALSE;
   STATUS[328].EXT.ModeBit3 := FALSE;
   STATUS[328].EXT.BIT19 := FALSE;
   STATUS[328].EXT.BIT20 := FALSE;
   STATUS[328].EXT.AlarmSuppressed := FALSE;
   STATUS[328].EXT.AlarmPrsent := FALSE;
   STATUS[328].EXT.AlarmFailUnAck := FALSE;
   STATUS[328].Status := 0;
   STATUS[328].TimeStamp := 16#0000;
   STATUS[329].VALUE := 0.0;
   STATUS[329].TRIGVALUE := 0.0;
   STATUS[329].EXT.AlarmWarnUnAck := FALSE;
   STATUS[329].EXT.AckRequired := FALSE;
   STATUS[329].EXT.Maintanence := FALSE;
   STATUS[329].EXT.Operation := FALSE;
   STATUS[329].EXT.Forced := FALSE;
   STATUS[329].EXT.BIT29 := FALSE;
   STATUS[329].EXT.BIT30 := FALSE;
   STATUS[329].EXT.BIT31 := FALSE;
   STATUS[329].EXT.ModeBit1 := FALSE;
   STATUS[329].EXT.ModeBit2 := FALSE;
   STATUS[329].EXT.ModeBit3 := FALSE;
   STATUS[329].EXT.BIT19 := FALSE;
   STATUS[329].EXT.BIT20 := FALSE;
   STATUS[329].EXT.AlarmSuppressed := FALSE;
   STATUS[329].EXT.AlarmPrsent := FALSE;
   STATUS[329].EXT.AlarmFailUnAck := FALSE;
   STATUS[329].Status := 0;
   STATUS[329].TimeStamp := 16#0000;
   STATUS[330].VALUE := 0.0;
   STATUS[330].TRIGVALUE := 0.0;
   STATUS[330].EXT.AlarmWarnUnAck := FALSE;
   STATUS[330].EXT.AckRequired := FALSE;
   STATUS[330].EXT.Maintanence := FALSE;
   STATUS[330].EXT.Operation := FALSE;
   STATUS[330].EXT.Forced := FALSE;
   STATUS[330].EXT.BIT29 := FALSE;
   STATUS[330].EXT.BIT30 := FALSE;
   STATUS[330].EXT.BIT31 := FALSE;
   STATUS[330].EXT.ModeBit1 := FALSE;
   STATUS[330].EXT.ModeBit2 := FALSE;
   STATUS[330].EXT.ModeBit3 := FALSE;
   STATUS[330].EXT.BIT19 := FALSE;
   STATUS[330].EXT.BIT20 := FALSE;
   STATUS[330].EXT.AlarmSuppressed := FALSE;
   STATUS[330].EXT.AlarmPrsent := FALSE;
   STATUS[330].EXT.AlarmFailUnAck := FALSE;
   STATUS[330].Status := 0;
   STATUS[330].TimeStamp := 16#0000;
   STATUS[331].VALUE := 0.0;
   STATUS[331].TRIGVALUE := 0.0;
   STATUS[331].EXT.AlarmWarnUnAck := FALSE;
   STATUS[331].EXT.AckRequired := FALSE;
   STATUS[331].EXT.Maintanence := FALSE;
   STATUS[331].EXT.Operation := FALSE;
   STATUS[331].EXT.Forced := FALSE;
   STATUS[331].EXT.BIT29 := FALSE;
   STATUS[331].EXT.BIT30 := FALSE;
   STATUS[331].EXT.BIT31 := FALSE;
   STATUS[331].EXT.ModeBit1 := FALSE;
   STATUS[331].EXT.ModeBit2 := FALSE;
   STATUS[331].EXT.ModeBit3 := FALSE;
   STATUS[331].EXT.BIT19 := FALSE;
   STATUS[331].EXT.BIT20 := FALSE;
   STATUS[331].EXT.AlarmSuppressed := FALSE;
   STATUS[331].EXT.AlarmPrsent := FALSE;
   STATUS[331].EXT.AlarmFailUnAck := FALSE;
   STATUS[331].Status := 0;
   STATUS[331].TimeStamp := 16#0000;
   STATUS[332].VALUE := 0.0;
   STATUS[332].TRIGVALUE := 0.0;
   STATUS[332].EXT.AlarmWarnUnAck := FALSE;
   STATUS[332].EXT.AckRequired := FALSE;
   STATUS[332].EXT.Maintanence := FALSE;
   STATUS[332].EXT.Operation := FALSE;
   STATUS[332].EXT.Forced := FALSE;
   STATUS[332].EXT.BIT29 := FALSE;
   STATUS[332].EXT.BIT30 := FALSE;
   STATUS[332].EXT.BIT31 := FALSE;
   STATUS[332].EXT.ModeBit1 := FALSE;
   STATUS[332].EXT.ModeBit2 := FALSE;
   STATUS[332].EXT.ModeBit3 := FALSE;
   STATUS[332].EXT.BIT19 := FALSE;
   STATUS[332].EXT.BIT20 := FALSE;
   STATUS[332].EXT.AlarmSuppressed := FALSE;
   STATUS[332].EXT.AlarmPrsent := FALSE;
   STATUS[332].EXT.AlarmFailUnAck := FALSE;
   STATUS[332].Status := 0;
   STATUS[332].TimeStamp := 16#0000;
   STATUS[333].VALUE := 0.0;
   STATUS[333].TRIGVALUE := 0.0;
   STATUS[333].EXT.AlarmWarnUnAck := FALSE;
   STATUS[333].EXT.AckRequired := FALSE;
   STATUS[333].EXT.Maintanence := FALSE;
   STATUS[333].EXT.Operation := FALSE;
   STATUS[333].EXT.Forced := FALSE;
   STATUS[333].EXT.BIT29 := FALSE;
   STATUS[333].EXT.BIT30 := FALSE;
   STATUS[333].EXT.BIT31 := FALSE;
   STATUS[333].EXT.ModeBit1 := FALSE;
   STATUS[333].EXT.ModeBit2 := FALSE;
   STATUS[333].EXT.ModeBit3 := FALSE;
   STATUS[333].EXT.BIT19 := FALSE;
   STATUS[333].EXT.BIT20 := FALSE;
   STATUS[333].EXT.AlarmSuppressed := FALSE;
   STATUS[333].EXT.AlarmPrsent := FALSE;
   STATUS[333].EXT.AlarmFailUnAck := FALSE;
   STATUS[333].Status := 0;
   STATUS[333].TimeStamp := 16#0000;
   STATUS[334].VALUE := 0.0;
   STATUS[334].TRIGVALUE := 0.0;
   STATUS[334].EXT.AlarmWarnUnAck := FALSE;
   STATUS[334].EXT.AckRequired := FALSE;
   STATUS[334].EXT.Maintanence := FALSE;
   STATUS[334].EXT.Operation := FALSE;
   STATUS[334].EXT.Forced := FALSE;
   STATUS[334].EXT.BIT29 := FALSE;
   STATUS[334].EXT.BIT30 := FALSE;
   STATUS[334].EXT.BIT31 := FALSE;
   STATUS[334].EXT.ModeBit1 := FALSE;
   STATUS[334].EXT.ModeBit2 := FALSE;
   STATUS[334].EXT.ModeBit3 := FALSE;
   STATUS[334].EXT.BIT19 := FALSE;
   STATUS[334].EXT.BIT20 := FALSE;
   STATUS[334].EXT.AlarmSuppressed := FALSE;
   STATUS[334].EXT.AlarmPrsent := FALSE;
   STATUS[334].EXT.AlarmFailUnAck := FALSE;
   STATUS[334].Status := 0;
   STATUS[334].TimeStamp := 16#0000;
   STATUS[335].VALUE := 0.0;
   STATUS[335].TRIGVALUE := 0.0;
   STATUS[335].EXT.AlarmWarnUnAck := FALSE;
   STATUS[335].EXT.AckRequired := FALSE;
   STATUS[335].EXT.Maintanence := FALSE;
   STATUS[335].EXT.Operation := FALSE;
   STATUS[335].EXT.Forced := FALSE;
   STATUS[335].EXT.BIT29 := FALSE;
   STATUS[335].EXT.BIT30 := FALSE;
   STATUS[335].EXT.BIT31 := FALSE;
   STATUS[335].EXT.ModeBit1 := FALSE;
   STATUS[335].EXT.ModeBit2 := FALSE;
   STATUS[335].EXT.ModeBit3 := FALSE;
   STATUS[335].EXT.BIT19 := FALSE;
   STATUS[335].EXT.BIT20 := FALSE;
   STATUS[335].EXT.AlarmSuppressed := FALSE;
   STATUS[335].EXT.AlarmPrsent := FALSE;
   STATUS[335].EXT.AlarmFailUnAck := FALSE;
   STATUS[335].Status := 0;
   STATUS[335].TimeStamp := 16#0000;
   STATUS[336].VALUE := 0.0;
   STATUS[336].TRIGVALUE := 0.0;
   STATUS[336].EXT.AlarmWarnUnAck := FALSE;
   STATUS[336].EXT.AckRequired := FALSE;
   STATUS[336].EXT.Maintanence := FALSE;
   STATUS[336].EXT.Operation := FALSE;
   STATUS[336].EXT.Forced := FALSE;
   STATUS[336].EXT.BIT29 := FALSE;
   STATUS[336].EXT.BIT30 := FALSE;
   STATUS[336].EXT.BIT31 := FALSE;
   STATUS[336].EXT.ModeBit1 := FALSE;
   STATUS[336].EXT.ModeBit2 := FALSE;
   STATUS[336].EXT.ModeBit3 := FALSE;
   STATUS[336].EXT.BIT19 := FALSE;
   STATUS[336].EXT.BIT20 := FALSE;
   STATUS[336].EXT.AlarmSuppressed := FALSE;
   STATUS[336].EXT.AlarmPrsent := FALSE;
   STATUS[336].EXT.AlarmFailUnAck := FALSE;
   STATUS[336].Status := 0;
   STATUS[336].TimeStamp := 16#0000;
   STATUS[337].VALUE := 0.0;
   STATUS[337].TRIGVALUE := 0.0;
   STATUS[337].EXT.AlarmWarnUnAck := FALSE;
   STATUS[337].EXT.AckRequired := FALSE;
   STATUS[337].EXT.Maintanence := FALSE;
   STATUS[337].EXT.Operation := FALSE;
   STATUS[337].EXT.Forced := FALSE;
   STATUS[337].EXT.BIT29 := FALSE;
   STATUS[337].EXT.BIT30 := FALSE;
   STATUS[337].EXT.BIT31 := FALSE;
   STATUS[337].EXT.ModeBit1 := FALSE;
   STATUS[337].EXT.ModeBit2 := FALSE;
   STATUS[337].EXT.ModeBit3 := FALSE;
   STATUS[337].EXT.BIT19 := FALSE;
   STATUS[337].EXT.BIT20 := FALSE;
   STATUS[337].EXT.AlarmSuppressed := FALSE;
   STATUS[337].EXT.AlarmPrsent := FALSE;
   STATUS[337].EXT.AlarmFailUnAck := FALSE;
   STATUS[337].Status := 0;
   STATUS[337].TimeStamp := 16#0000;
   STATUS[338].VALUE := 0.0;
   STATUS[338].TRIGVALUE := 0.0;
   STATUS[338].EXT.AlarmWarnUnAck := FALSE;
   STATUS[338].EXT.AckRequired := FALSE;
   STATUS[338].EXT.Maintanence := FALSE;
   STATUS[338].EXT.Operation := FALSE;
   STATUS[338].EXT.Forced := FALSE;
   STATUS[338].EXT.BIT29 := FALSE;
   STATUS[338].EXT.BIT30 := FALSE;
   STATUS[338].EXT.BIT31 := FALSE;
   STATUS[338].EXT.ModeBit1 := FALSE;
   STATUS[338].EXT.ModeBit2 := FALSE;
   STATUS[338].EXT.ModeBit3 := FALSE;
   STATUS[338].EXT.BIT19 := FALSE;
   STATUS[338].EXT.BIT20 := FALSE;
   STATUS[338].EXT.AlarmSuppressed := FALSE;
   STATUS[338].EXT.AlarmPrsent := FALSE;
   STATUS[338].EXT.AlarmFailUnAck := FALSE;
   STATUS[338].Status := 0;
   STATUS[338].TimeStamp := 16#0000;
   STATUS[339].VALUE := 0.0;
   STATUS[339].TRIGVALUE := 0.0;
   STATUS[339].EXT.AlarmWarnUnAck := FALSE;
   STATUS[339].EXT.AckRequired := FALSE;
   STATUS[339].EXT.Maintanence := FALSE;
   STATUS[339].EXT.Operation := FALSE;
   STATUS[339].EXT.Forced := FALSE;
   STATUS[339].EXT.BIT29 := FALSE;
   STATUS[339].EXT.BIT30 := FALSE;
   STATUS[339].EXT.BIT31 := FALSE;
   STATUS[339].EXT.ModeBit1 := FALSE;
   STATUS[339].EXT.ModeBit2 := FALSE;
   STATUS[339].EXT.ModeBit3 := FALSE;
   STATUS[339].EXT.BIT19 := FALSE;
   STATUS[339].EXT.BIT20 := FALSE;
   STATUS[339].EXT.AlarmSuppressed := FALSE;
   STATUS[339].EXT.AlarmPrsent := FALSE;
   STATUS[339].EXT.AlarmFailUnAck := FALSE;
   STATUS[339].Status := 0;
   STATUS[339].TimeStamp := 16#0000;
   STATUS[340].VALUE := 0.0;
   STATUS[340].TRIGVALUE := 0.0;
   STATUS[340].EXT.AlarmWarnUnAck := FALSE;
   STATUS[340].EXT.AckRequired := FALSE;
   STATUS[340].EXT.Maintanence := FALSE;
   STATUS[340].EXT.Operation := FALSE;
   STATUS[340].EXT.Forced := FALSE;
   STATUS[340].EXT.BIT29 := FALSE;
   STATUS[340].EXT.BIT30 := FALSE;
   STATUS[340].EXT.BIT31 := FALSE;
   STATUS[340].EXT.ModeBit1 := FALSE;
   STATUS[340].EXT.ModeBit2 := FALSE;
   STATUS[340].EXT.ModeBit3 := FALSE;
   STATUS[340].EXT.BIT19 := FALSE;
   STATUS[340].EXT.BIT20 := FALSE;
   STATUS[340].EXT.AlarmSuppressed := FALSE;
   STATUS[340].EXT.AlarmPrsent := FALSE;
   STATUS[340].EXT.AlarmFailUnAck := FALSE;
   STATUS[340].Status := 0;
   STATUS[340].TimeStamp := 16#0000;
   STATUS[341].VALUE := 0.0;
   STATUS[341].TRIGVALUE := 0.0;
   STATUS[341].EXT.AlarmWarnUnAck := FALSE;
   STATUS[341].EXT.AckRequired := FALSE;
   STATUS[341].EXT.Maintanence := FALSE;
   STATUS[341].EXT.Operation := FALSE;
   STATUS[341].EXT.Forced := FALSE;
   STATUS[341].EXT.BIT29 := FALSE;
   STATUS[341].EXT.BIT30 := FALSE;
   STATUS[341].EXT.BIT31 := FALSE;
   STATUS[341].EXT.ModeBit1 := FALSE;
   STATUS[341].EXT.ModeBit2 := FALSE;
   STATUS[341].EXT.ModeBit3 := FALSE;
   STATUS[341].EXT.BIT19 := FALSE;
   STATUS[341].EXT.BIT20 := FALSE;
   STATUS[341].EXT.AlarmSuppressed := FALSE;
   STATUS[341].EXT.AlarmPrsent := FALSE;
   STATUS[341].EXT.AlarmFailUnAck := FALSE;
   STATUS[341].Status := 0;
   STATUS[341].TimeStamp := 16#0000;
   STATUS[342].VALUE := 0.0;
   STATUS[342].TRIGVALUE := 0.0;
   STATUS[342].EXT.AlarmWarnUnAck := FALSE;
   STATUS[342].EXT.AckRequired := FALSE;
   STATUS[342].EXT.Maintanence := FALSE;
   STATUS[342].EXT.Operation := FALSE;
   STATUS[342].EXT.Forced := FALSE;
   STATUS[342].EXT.BIT29 := FALSE;
   STATUS[342].EXT.BIT30 := FALSE;
   STATUS[342].EXT.BIT31 := FALSE;
   STATUS[342].EXT.ModeBit1 := FALSE;
   STATUS[342].EXT.ModeBit2 := FALSE;
   STATUS[342].EXT.ModeBit3 := FALSE;
   STATUS[342].EXT.BIT19 := FALSE;
   STATUS[342].EXT.BIT20 := FALSE;
   STATUS[342].EXT.AlarmSuppressed := FALSE;
   STATUS[342].EXT.AlarmPrsent := FALSE;
   STATUS[342].EXT.AlarmFailUnAck := FALSE;
   STATUS[342].Status := 0;
   STATUS[342].TimeStamp := 16#0000;
   STATUS[343].VALUE := 0.0;
   STATUS[343].TRIGVALUE := 0.0;
   STATUS[343].EXT.AlarmWarnUnAck := FALSE;
   STATUS[343].EXT.AckRequired := FALSE;
   STATUS[343].EXT.Maintanence := FALSE;
   STATUS[343].EXT.Operation := FALSE;
   STATUS[343].EXT.Forced := FALSE;
   STATUS[343].EXT.BIT29 := FALSE;
   STATUS[343].EXT.BIT30 := FALSE;
   STATUS[343].EXT.BIT31 := FALSE;
   STATUS[343].EXT.ModeBit1 := FALSE;
   STATUS[343].EXT.ModeBit2 := FALSE;
   STATUS[343].EXT.ModeBit3 := FALSE;
   STATUS[343].EXT.BIT19 := FALSE;
   STATUS[343].EXT.BIT20 := FALSE;
   STATUS[343].EXT.AlarmSuppressed := FALSE;
   STATUS[343].EXT.AlarmPrsent := FALSE;
   STATUS[343].EXT.AlarmFailUnAck := FALSE;
   STATUS[343].Status := 0;
   STATUS[343].TimeStamp := 16#0000;
   STATUS[344].VALUE := 0.0;
   STATUS[344].TRIGVALUE := 0.0;
   STATUS[344].EXT.AlarmWarnUnAck := FALSE;
   STATUS[344].EXT.AckRequired := FALSE;
   STATUS[344].EXT.Maintanence := FALSE;
   STATUS[344].EXT.Operation := FALSE;
   STATUS[344].EXT.Forced := FALSE;
   STATUS[344].EXT.BIT29 := FALSE;
   STATUS[344].EXT.BIT30 := FALSE;
   STATUS[344].EXT.BIT31 := FALSE;
   STATUS[344].EXT.ModeBit1 := FALSE;
   STATUS[344].EXT.ModeBit2 := FALSE;
   STATUS[344].EXT.ModeBit3 := FALSE;
   STATUS[344].EXT.BIT19 := FALSE;
   STATUS[344].EXT.BIT20 := FALSE;
   STATUS[344].EXT.AlarmSuppressed := FALSE;
   STATUS[344].EXT.AlarmPrsent := FALSE;
   STATUS[344].EXT.AlarmFailUnAck := FALSE;
   STATUS[344].Status := 0;
   STATUS[344].TimeStamp := 16#0000;
   STATUS[345].VALUE := 0.0;
   STATUS[345].TRIGVALUE := 0.0;
   STATUS[345].EXT.AlarmWarnUnAck := FALSE;
   STATUS[345].EXT.AckRequired := FALSE;
   STATUS[345].EXT.Maintanence := FALSE;
   STATUS[345].EXT.Operation := FALSE;
   STATUS[345].EXT.Forced := FALSE;
   STATUS[345].EXT.BIT29 := FALSE;
   STATUS[345].EXT.BIT30 := FALSE;
   STATUS[345].EXT.BIT31 := FALSE;
   STATUS[345].EXT.ModeBit1 := FALSE;
   STATUS[345].EXT.ModeBit2 := FALSE;
   STATUS[345].EXT.ModeBit3 := FALSE;
   STATUS[345].EXT.BIT19 := FALSE;
   STATUS[345].EXT.BIT20 := FALSE;
   STATUS[345].EXT.AlarmSuppressed := FALSE;
   STATUS[345].EXT.AlarmPrsent := FALSE;
   STATUS[345].EXT.AlarmFailUnAck := FALSE;
   STATUS[345].Status := 0;
   STATUS[345].TimeStamp := 16#0000;
   STATUS[346].VALUE := 0.0;
   STATUS[346].TRIGVALUE := 0.0;
   STATUS[346].EXT.AlarmWarnUnAck := FALSE;
   STATUS[346].EXT.AckRequired := FALSE;
   STATUS[346].EXT.Maintanence := FALSE;
   STATUS[346].EXT.Operation := FALSE;
   STATUS[346].EXT.Forced := FALSE;
   STATUS[346].EXT.BIT29 := FALSE;
   STATUS[346].EXT.BIT30 := FALSE;
   STATUS[346].EXT.BIT31 := FALSE;
   STATUS[346].EXT.ModeBit1 := FALSE;
   STATUS[346].EXT.ModeBit2 := FALSE;
   STATUS[346].EXT.ModeBit3 := FALSE;
   STATUS[346].EXT.BIT19 := FALSE;
   STATUS[346].EXT.BIT20 := FALSE;
   STATUS[346].EXT.AlarmSuppressed := FALSE;
   STATUS[346].EXT.AlarmPrsent := FALSE;
   STATUS[346].EXT.AlarmFailUnAck := FALSE;
   STATUS[346].Status := 0;
   STATUS[346].TimeStamp := 16#0000;
   STATUS[347].VALUE := 0.0;
   STATUS[347].TRIGVALUE := 0.0;
   STATUS[347].EXT.AlarmWarnUnAck := FALSE;
   STATUS[347].EXT.AckRequired := FALSE;
   STATUS[347].EXT.Maintanence := FALSE;
   STATUS[347].EXT.Operation := FALSE;
   STATUS[347].EXT.Forced := FALSE;
   STATUS[347].EXT.BIT29 := FALSE;
   STATUS[347].EXT.BIT30 := FALSE;
   STATUS[347].EXT.BIT31 := FALSE;
   STATUS[347].EXT.ModeBit1 := FALSE;
   STATUS[347].EXT.ModeBit2 := FALSE;
   STATUS[347].EXT.ModeBit3 := FALSE;
   STATUS[347].EXT.BIT19 := FALSE;
   STATUS[347].EXT.BIT20 := FALSE;
   STATUS[347].EXT.AlarmSuppressed := FALSE;
   STATUS[347].EXT.AlarmPrsent := FALSE;
   STATUS[347].EXT.AlarmFailUnAck := FALSE;
   STATUS[347].Status := 0;
   STATUS[347].TimeStamp := 16#0000;
   STATUS[348].VALUE := 0.0;
   STATUS[348].TRIGVALUE := 0.0;
   STATUS[348].EXT.AlarmWarnUnAck := FALSE;
   STATUS[348].EXT.AckRequired := FALSE;
   STATUS[348].EXT.Maintanence := FALSE;
   STATUS[348].EXT.Operation := FALSE;
   STATUS[348].EXT.Forced := FALSE;
   STATUS[348].EXT.BIT29 := FALSE;
   STATUS[348].EXT.BIT30 := FALSE;
   STATUS[348].EXT.BIT31 := FALSE;
   STATUS[348].EXT.ModeBit1 := FALSE;
   STATUS[348].EXT.ModeBit2 := FALSE;
   STATUS[348].EXT.ModeBit3 := FALSE;
   STATUS[348].EXT.BIT19 := FALSE;
   STATUS[348].EXT.BIT20 := FALSE;
   STATUS[348].EXT.AlarmSuppressed := FALSE;
   STATUS[348].EXT.AlarmPrsent := FALSE;
   STATUS[348].EXT.AlarmFailUnAck := FALSE;
   STATUS[348].Status := 0;
   STATUS[348].TimeStamp := 16#0000;
   STATUS[349].VALUE := 0.0;
   STATUS[349].TRIGVALUE := 0.0;
   STATUS[349].EXT.AlarmWarnUnAck := FALSE;
   STATUS[349].EXT.AckRequired := FALSE;
   STATUS[349].EXT.Maintanence := FALSE;
   STATUS[349].EXT.Operation := FALSE;
   STATUS[349].EXT.Forced := FALSE;
   STATUS[349].EXT.BIT29 := FALSE;
   STATUS[349].EXT.BIT30 := FALSE;
   STATUS[349].EXT.BIT31 := FALSE;
   STATUS[349].EXT.ModeBit1 := FALSE;
   STATUS[349].EXT.ModeBit2 := FALSE;
   STATUS[349].EXT.ModeBit3 := FALSE;
   STATUS[349].EXT.BIT19 := FALSE;
   STATUS[349].EXT.BIT20 := FALSE;
   STATUS[349].EXT.AlarmSuppressed := FALSE;
   STATUS[349].EXT.AlarmPrsent := FALSE;
   STATUS[349].EXT.AlarmFailUnAck := FALSE;
   STATUS[349].Status := 0;
   STATUS[349].TimeStamp := 16#0000;
   STATUS[350].VALUE := 0.0;
   STATUS[350].TRIGVALUE := 0.0;
   STATUS[350].EXT.AlarmWarnUnAck := FALSE;
   STATUS[350].EXT.AckRequired := FALSE;
   STATUS[350].EXT.Maintanence := FALSE;
   STATUS[350].EXT.Operation := FALSE;
   STATUS[350].EXT.Forced := FALSE;
   STATUS[350].EXT.BIT29 := FALSE;
   STATUS[350].EXT.BIT30 := FALSE;
   STATUS[350].EXT.BIT31 := FALSE;
   STATUS[350].EXT.ModeBit1 := FALSE;
   STATUS[350].EXT.ModeBit2 := FALSE;
   STATUS[350].EXT.ModeBit3 := FALSE;
   STATUS[350].EXT.BIT19 := FALSE;
   STATUS[350].EXT.BIT20 := FALSE;
   STATUS[350].EXT.AlarmSuppressed := FALSE;
   STATUS[350].EXT.AlarmPrsent := FALSE;
   STATUS[350].EXT.AlarmFailUnAck := FALSE;
   STATUS[350].Status := 0;
   STATUS[350].TimeStamp := 16#0000;
   STATUS[351].VALUE := 0.0;
   STATUS[351].TRIGVALUE := 0.0;
   STATUS[351].EXT.AlarmWarnUnAck := FALSE;
   STATUS[351].EXT.AckRequired := FALSE;
   STATUS[351].EXT.Maintanence := FALSE;
   STATUS[351].EXT.Operation := FALSE;
   STATUS[351].EXT.Forced := FALSE;
   STATUS[351].EXT.BIT29 := FALSE;
   STATUS[351].EXT.BIT30 := FALSE;
   STATUS[351].EXT.BIT31 := FALSE;
   STATUS[351].EXT.ModeBit1 := FALSE;
   STATUS[351].EXT.ModeBit2 := FALSE;
   STATUS[351].EXT.ModeBit3 := FALSE;
   STATUS[351].EXT.BIT19 := FALSE;
   STATUS[351].EXT.BIT20 := FALSE;
   STATUS[351].EXT.AlarmSuppressed := FALSE;
   STATUS[351].EXT.AlarmPrsent := FALSE;
   STATUS[351].EXT.AlarmFailUnAck := FALSE;
   STATUS[351].Status := 0;
   STATUS[351].TimeStamp := 16#0000;
   STATUS[352].VALUE := 0.0;
   STATUS[352].TRIGVALUE := 0.0;
   STATUS[352].EXT.AlarmWarnUnAck := FALSE;
   STATUS[352].EXT.AckRequired := FALSE;
   STATUS[352].EXT.Maintanence := FALSE;
   STATUS[352].EXT.Operation := FALSE;
   STATUS[352].EXT.Forced := FALSE;
   STATUS[352].EXT.BIT29 := FALSE;
   STATUS[352].EXT.BIT30 := FALSE;
   STATUS[352].EXT.BIT31 := FALSE;
   STATUS[352].EXT.ModeBit1 := FALSE;
   STATUS[352].EXT.ModeBit2 := FALSE;
   STATUS[352].EXT.ModeBit3 := FALSE;
   STATUS[352].EXT.BIT19 := FALSE;
   STATUS[352].EXT.BIT20 := FALSE;
   STATUS[352].EXT.AlarmSuppressed := FALSE;
   STATUS[352].EXT.AlarmPrsent := FALSE;
   STATUS[352].EXT.AlarmFailUnAck := FALSE;
   STATUS[352].Status := 0;
   STATUS[352].TimeStamp := 16#0000;
   STATUS[353].VALUE := 0.0;
   STATUS[353].TRIGVALUE := 0.0;
   STATUS[353].EXT.AlarmWarnUnAck := FALSE;
   STATUS[353].EXT.AckRequired := FALSE;
   STATUS[353].EXT.Maintanence := FALSE;
   STATUS[353].EXT.Operation := FALSE;
   STATUS[353].EXT.Forced := FALSE;
   STATUS[353].EXT.BIT29 := FALSE;
   STATUS[353].EXT.BIT30 := FALSE;
   STATUS[353].EXT.BIT31 := FALSE;
   STATUS[353].EXT.ModeBit1 := FALSE;
   STATUS[353].EXT.ModeBit2 := FALSE;
   STATUS[353].EXT.ModeBit3 := FALSE;
   STATUS[353].EXT.BIT19 := FALSE;
   STATUS[353].EXT.BIT20 := FALSE;
   STATUS[353].EXT.AlarmSuppressed := FALSE;
   STATUS[353].EXT.AlarmPrsent := FALSE;
   STATUS[353].EXT.AlarmFailUnAck := FALSE;
   STATUS[353].Status := 0;
   STATUS[353].TimeStamp := 16#0000;
   STATUS[354].VALUE := 0.0;
   STATUS[354].TRIGVALUE := 0.0;
   STATUS[354].EXT.AlarmWarnUnAck := FALSE;
   STATUS[354].EXT.AckRequired := FALSE;
   STATUS[354].EXT.Maintanence := FALSE;
   STATUS[354].EXT.Operation := FALSE;
   STATUS[354].EXT.Forced := FALSE;
   STATUS[354].EXT.BIT29 := FALSE;
   STATUS[354].EXT.BIT30 := FALSE;
   STATUS[354].EXT.BIT31 := FALSE;
   STATUS[354].EXT.ModeBit1 := FALSE;
   STATUS[354].EXT.ModeBit2 := FALSE;
   STATUS[354].EXT.ModeBit3 := FALSE;
   STATUS[354].EXT.BIT19 := FALSE;
   STATUS[354].EXT.BIT20 := FALSE;
   STATUS[354].EXT.AlarmSuppressed := FALSE;
   STATUS[354].EXT.AlarmPrsent := FALSE;
   STATUS[354].EXT.AlarmFailUnAck := FALSE;
   STATUS[354].Status := 0;
   STATUS[354].TimeStamp := 16#0000;
   STATUS[355].VALUE := 0.0;
   STATUS[355].TRIGVALUE := 0.0;
   STATUS[355].EXT.AlarmWarnUnAck := FALSE;
   STATUS[355].EXT.AckRequired := FALSE;
   STATUS[355].EXT.Maintanence := FALSE;
   STATUS[355].EXT.Operation := FALSE;
   STATUS[355].EXT.Forced := FALSE;
   STATUS[355].EXT.BIT29 := FALSE;
   STATUS[355].EXT.BIT30 := FALSE;
   STATUS[355].EXT.BIT31 := FALSE;
   STATUS[355].EXT.ModeBit1 := FALSE;
   STATUS[355].EXT.ModeBit2 := FALSE;
   STATUS[355].EXT.ModeBit3 := FALSE;
   STATUS[355].EXT.BIT19 := FALSE;
   STATUS[355].EXT.BIT20 := FALSE;
   STATUS[355].EXT.AlarmSuppressed := FALSE;
   STATUS[355].EXT.AlarmPrsent := FALSE;
   STATUS[355].EXT.AlarmFailUnAck := FALSE;
   STATUS[355].Status := 0;
   STATUS[355].TimeStamp := 16#0000;
   STATUS[356].VALUE := 0.0;
   STATUS[356].TRIGVALUE := 0.0;
   STATUS[356].EXT.AlarmWarnUnAck := FALSE;
   STATUS[356].EXT.AckRequired := FALSE;
   STATUS[356].EXT.Maintanence := FALSE;
   STATUS[356].EXT.Operation := FALSE;
   STATUS[356].EXT.Forced := FALSE;
   STATUS[356].EXT.BIT29 := FALSE;
   STATUS[356].EXT.BIT30 := FALSE;
   STATUS[356].EXT.BIT31 := FALSE;
   STATUS[356].EXT.ModeBit1 := FALSE;
   STATUS[356].EXT.ModeBit2 := FALSE;
   STATUS[356].EXT.ModeBit3 := FALSE;
   STATUS[356].EXT.BIT19 := FALSE;
   STATUS[356].EXT.BIT20 := FALSE;
   STATUS[356].EXT.AlarmSuppressed := FALSE;
   STATUS[356].EXT.AlarmPrsent := FALSE;
   STATUS[356].EXT.AlarmFailUnAck := FALSE;
   STATUS[356].Status := 0;
   STATUS[356].TimeStamp := 16#0000;
   STATUS[357].VALUE := 0.0;
   STATUS[357].TRIGVALUE := 0.0;
   STATUS[357].EXT.AlarmWarnUnAck := FALSE;
   STATUS[357].EXT.AckRequired := FALSE;
   STATUS[357].EXT.Maintanence := FALSE;
   STATUS[357].EXT.Operation := FALSE;
   STATUS[357].EXT.Forced := FALSE;
   STATUS[357].EXT.BIT29 := FALSE;
   STATUS[357].EXT.BIT30 := FALSE;
   STATUS[357].EXT.BIT31 := FALSE;
   STATUS[357].EXT.ModeBit1 := FALSE;
   STATUS[357].EXT.ModeBit2 := FALSE;
   STATUS[357].EXT.ModeBit3 := FALSE;
   STATUS[357].EXT.BIT19 := FALSE;
   STATUS[357].EXT.BIT20 := FALSE;
   STATUS[357].EXT.AlarmSuppressed := FALSE;
   STATUS[357].EXT.AlarmPrsent := FALSE;
   STATUS[357].EXT.AlarmFailUnAck := FALSE;
   STATUS[357].Status := 0;
   STATUS[357].TimeStamp := 16#0000;
   STATUS[358].VALUE := 0.0;
   STATUS[358].TRIGVALUE := 0.0;
   STATUS[358].EXT.AlarmWarnUnAck := FALSE;
   STATUS[358].EXT.AckRequired := FALSE;
   STATUS[358].EXT.Maintanence := FALSE;
   STATUS[358].EXT.Operation := FALSE;
   STATUS[358].EXT.Forced := FALSE;
   STATUS[358].EXT.BIT29 := FALSE;
   STATUS[358].EXT.BIT30 := FALSE;
   STATUS[358].EXT.BIT31 := FALSE;
   STATUS[358].EXT.ModeBit1 := FALSE;
   STATUS[358].EXT.ModeBit2 := FALSE;
   STATUS[358].EXT.ModeBit3 := FALSE;
   STATUS[358].EXT.BIT19 := FALSE;
   STATUS[358].EXT.BIT20 := FALSE;
   STATUS[358].EXT.AlarmSuppressed := FALSE;
   STATUS[358].EXT.AlarmPrsent := FALSE;
   STATUS[358].EXT.AlarmFailUnAck := FALSE;
   STATUS[358].Status := 0;
   STATUS[358].TimeStamp := 16#0000;
   STATUS[359].VALUE := 0.0;
   STATUS[359].TRIGVALUE := 0.0;
   STATUS[359].EXT.AlarmWarnUnAck := FALSE;
   STATUS[359].EXT.AckRequired := FALSE;
   STATUS[359].EXT.Maintanence := FALSE;
   STATUS[359].EXT.Operation := FALSE;
   STATUS[359].EXT.Forced := FALSE;
   STATUS[359].EXT.BIT29 := FALSE;
   STATUS[359].EXT.BIT30 := FALSE;
   STATUS[359].EXT.BIT31 := FALSE;
   STATUS[359].EXT.ModeBit1 := FALSE;
   STATUS[359].EXT.ModeBit2 := FALSE;
   STATUS[359].EXT.ModeBit3 := FALSE;
   STATUS[359].EXT.BIT19 := FALSE;
   STATUS[359].EXT.BIT20 := FALSE;
   STATUS[359].EXT.AlarmSuppressed := FALSE;
   STATUS[359].EXT.AlarmPrsent := FALSE;
   STATUS[359].EXT.AlarmFailUnAck := FALSE;
   STATUS[359].Status := 0;
   STATUS[359].TimeStamp := 16#0000;
   STATUS[360].VALUE := 0.0;
   STATUS[360].TRIGVALUE := 0.0;
   STATUS[360].EXT.AlarmWarnUnAck := FALSE;
   STATUS[360].EXT.AckRequired := FALSE;
   STATUS[360].EXT.Maintanence := FALSE;
   STATUS[360].EXT.Operation := FALSE;
   STATUS[360].EXT.Forced := FALSE;
   STATUS[360].EXT.BIT29 := FALSE;
   STATUS[360].EXT.BIT30 := FALSE;
   STATUS[360].EXT.BIT31 := FALSE;
   STATUS[360].EXT.ModeBit1 := FALSE;
   STATUS[360].EXT.ModeBit2 := FALSE;
   STATUS[360].EXT.ModeBit3 := FALSE;
   STATUS[360].EXT.BIT19 := FALSE;
   STATUS[360].EXT.BIT20 := FALSE;
   STATUS[360].EXT.AlarmSuppressed := FALSE;
   STATUS[360].EXT.AlarmPrsent := FALSE;
   STATUS[360].EXT.AlarmFailUnAck := FALSE;
   STATUS[360].Status := 0;
   STATUS[360].TimeStamp := 16#0000;
   STATUS[361].VALUE := 0.0;
   STATUS[361].TRIGVALUE := 0.0;
   STATUS[361].EXT.AlarmWarnUnAck := FALSE;
   STATUS[361].EXT.AckRequired := FALSE;
   STATUS[361].EXT.Maintanence := FALSE;
   STATUS[361].EXT.Operation := FALSE;
   STATUS[361].EXT.Forced := FALSE;
   STATUS[361].EXT.BIT29 := FALSE;
   STATUS[361].EXT.BIT30 := FALSE;
   STATUS[361].EXT.BIT31 := FALSE;
   STATUS[361].EXT.ModeBit1 := FALSE;
   STATUS[361].EXT.ModeBit2 := FALSE;
   STATUS[361].EXT.ModeBit3 := FALSE;
   STATUS[361].EXT.BIT19 := FALSE;
   STATUS[361].EXT.BIT20 := FALSE;
   STATUS[361].EXT.AlarmSuppressed := FALSE;
   STATUS[361].EXT.AlarmPrsent := FALSE;
   STATUS[361].EXT.AlarmFailUnAck := FALSE;
   STATUS[361].Status := 0;
   STATUS[361].TimeStamp := 16#0000;
   STATUS[362].VALUE := 0.0;
   STATUS[362].TRIGVALUE := 0.0;
   STATUS[362].EXT.AlarmWarnUnAck := FALSE;
   STATUS[362].EXT.AckRequired := FALSE;
   STATUS[362].EXT.Maintanence := FALSE;
   STATUS[362].EXT.Operation := FALSE;
   STATUS[362].EXT.Forced := FALSE;
   STATUS[362].EXT.BIT29 := FALSE;
   STATUS[362].EXT.BIT30 := FALSE;
   STATUS[362].EXT.BIT31 := FALSE;
   STATUS[362].EXT.ModeBit1 := FALSE;
   STATUS[362].EXT.ModeBit2 := FALSE;
   STATUS[362].EXT.ModeBit3 := FALSE;
   STATUS[362].EXT.BIT19 := FALSE;
   STATUS[362].EXT.BIT20 := FALSE;
   STATUS[362].EXT.AlarmSuppressed := FALSE;
   STATUS[362].EXT.AlarmPrsent := FALSE;
   STATUS[362].EXT.AlarmFailUnAck := FALSE;
   STATUS[362].Status := 0;
   STATUS[362].TimeStamp := 16#0000;
   STATUS[363].VALUE := 0.0;
   STATUS[363].TRIGVALUE := 0.0;
   STATUS[363].EXT.AlarmWarnUnAck := FALSE;
   STATUS[363].EXT.AckRequired := FALSE;
   STATUS[363].EXT.Maintanence := FALSE;
   STATUS[363].EXT.Operation := FALSE;
   STATUS[363].EXT.Forced := FALSE;
   STATUS[363].EXT.BIT29 := FALSE;
   STATUS[363].EXT.BIT30 := FALSE;
   STATUS[363].EXT.BIT31 := FALSE;
   STATUS[363].EXT.ModeBit1 := FALSE;
   STATUS[363].EXT.ModeBit2 := FALSE;
   STATUS[363].EXT.ModeBit3 := FALSE;
   STATUS[363].EXT.BIT19 := FALSE;
   STATUS[363].EXT.BIT20 := FALSE;
   STATUS[363].EXT.AlarmSuppressed := FALSE;
   STATUS[363].EXT.AlarmPrsent := FALSE;
   STATUS[363].EXT.AlarmFailUnAck := FALSE;
   STATUS[363].Status := 0;
   STATUS[363].TimeStamp := 16#0000;
   STATUS[364].VALUE := 0.0;
   STATUS[364].TRIGVALUE := 0.0;
   STATUS[364].EXT.AlarmWarnUnAck := FALSE;
   STATUS[364].EXT.AckRequired := FALSE;
   STATUS[364].EXT.Maintanence := FALSE;
   STATUS[364].EXT.Operation := FALSE;
   STATUS[364].EXT.Forced := FALSE;
   STATUS[364].EXT.BIT29 := FALSE;
   STATUS[364].EXT.BIT30 := FALSE;
   STATUS[364].EXT.BIT31 := FALSE;
   STATUS[364].EXT.ModeBit1 := FALSE;
   STATUS[364].EXT.ModeBit2 := FALSE;
   STATUS[364].EXT.ModeBit3 := FALSE;
   STATUS[364].EXT.BIT19 := FALSE;
   STATUS[364].EXT.BIT20 := FALSE;
   STATUS[364].EXT.AlarmSuppressed := FALSE;
   STATUS[364].EXT.AlarmPrsent := FALSE;
   STATUS[364].EXT.AlarmFailUnAck := FALSE;
   STATUS[364].Status := 0;
   STATUS[364].TimeStamp := 16#0000;
   STATUS[365].VALUE := 0.0;
   STATUS[365].TRIGVALUE := 0.0;
   STATUS[365].EXT.AlarmWarnUnAck := FALSE;
   STATUS[365].EXT.AckRequired := FALSE;
   STATUS[365].EXT.Maintanence := FALSE;
   STATUS[365].EXT.Operation := FALSE;
   STATUS[365].EXT.Forced := FALSE;
   STATUS[365].EXT.BIT29 := FALSE;
   STATUS[365].EXT.BIT30 := FALSE;
   STATUS[365].EXT.BIT31 := FALSE;
   STATUS[365].EXT.ModeBit1 := FALSE;
   STATUS[365].EXT.ModeBit2 := FALSE;
   STATUS[365].EXT.ModeBit3 := FALSE;
   STATUS[365].EXT.BIT19 := FALSE;
   STATUS[365].EXT.BIT20 := FALSE;
   STATUS[365].EXT.AlarmSuppressed := FALSE;
   STATUS[365].EXT.AlarmPrsent := FALSE;
   STATUS[365].EXT.AlarmFailUnAck := FALSE;
   STATUS[365].Status := 0;
   STATUS[365].TimeStamp := 16#0000;
   STATUS[366].VALUE := 0.0;
   STATUS[366].TRIGVALUE := 0.0;
   STATUS[366].EXT.AlarmWarnUnAck := FALSE;
   STATUS[366].EXT.AckRequired := FALSE;
   STATUS[366].EXT.Maintanence := FALSE;
   STATUS[366].EXT.Operation := FALSE;
   STATUS[366].EXT.Forced := FALSE;
   STATUS[366].EXT.BIT29 := FALSE;
   STATUS[366].EXT.BIT30 := FALSE;
   STATUS[366].EXT.BIT31 := FALSE;
   STATUS[366].EXT.ModeBit1 := FALSE;
   STATUS[366].EXT.ModeBit2 := FALSE;
   STATUS[366].EXT.ModeBit3 := FALSE;
   STATUS[366].EXT.BIT19 := FALSE;
   STATUS[366].EXT.BIT20 := FALSE;
   STATUS[366].EXT.AlarmSuppressed := FALSE;
   STATUS[366].EXT.AlarmPrsent := FALSE;
   STATUS[366].EXT.AlarmFailUnAck := FALSE;
   STATUS[366].Status := 0;
   STATUS[366].TimeStamp := 16#0000;
   STATUS[367].VALUE := 0.0;
   STATUS[367].TRIGVALUE := 0.0;
   STATUS[367].EXT.AlarmWarnUnAck := FALSE;
   STATUS[367].EXT.AckRequired := FALSE;
   STATUS[367].EXT.Maintanence := FALSE;
   STATUS[367].EXT.Operation := FALSE;
   STATUS[367].EXT.Forced := FALSE;
   STATUS[367].EXT.BIT29 := FALSE;
   STATUS[367].EXT.BIT30 := FALSE;
   STATUS[367].EXT.BIT31 := FALSE;
   STATUS[367].EXT.ModeBit1 := FALSE;
   STATUS[367].EXT.ModeBit2 := FALSE;
   STATUS[367].EXT.ModeBit3 := FALSE;
   STATUS[367].EXT.BIT19 := FALSE;
   STATUS[367].EXT.BIT20 := FALSE;
   STATUS[367].EXT.AlarmSuppressed := FALSE;
   STATUS[367].EXT.AlarmPrsent := FALSE;
   STATUS[367].EXT.AlarmFailUnAck := FALSE;
   STATUS[367].Status := 0;
   STATUS[367].TimeStamp := 16#0000;
   STATUS[368].VALUE := 0.0;
   STATUS[368].TRIGVALUE := 0.0;
   STATUS[368].EXT.AlarmWarnUnAck := FALSE;
   STATUS[368].EXT.AckRequired := FALSE;
   STATUS[368].EXT.Maintanence := FALSE;
   STATUS[368].EXT.Operation := FALSE;
   STATUS[368].EXT.Forced := FALSE;
   STATUS[368].EXT.BIT29 := FALSE;
   STATUS[368].EXT.BIT30 := FALSE;
   STATUS[368].EXT.BIT31 := FALSE;
   STATUS[368].EXT.ModeBit1 := FALSE;
   STATUS[368].EXT.ModeBit2 := FALSE;
   STATUS[368].EXT.ModeBit3 := FALSE;
   STATUS[368].EXT.BIT19 := FALSE;
   STATUS[368].EXT.BIT20 := FALSE;
   STATUS[368].EXT.AlarmSuppressed := FALSE;
   STATUS[368].EXT.AlarmPrsent := FALSE;
   STATUS[368].EXT.AlarmFailUnAck := FALSE;
   STATUS[368].Status := 0;
   STATUS[368].TimeStamp := 16#0000;
   STATUS[369].VALUE := 0.0;
   STATUS[369].TRIGVALUE := 0.0;
   STATUS[369].EXT.AlarmWarnUnAck := FALSE;
   STATUS[369].EXT.AckRequired := FALSE;
   STATUS[369].EXT.Maintanence := FALSE;
   STATUS[369].EXT.Operation := FALSE;
   STATUS[369].EXT.Forced := FALSE;
   STATUS[369].EXT.BIT29 := FALSE;
   STATUS[369].EXT.BIT30 := FALSE;
   STATUS[369].EXT.BIT31 := FALSE;
   STATUS[369].EXT.ModeBit1 := FALSE;
   STATUS[369].EXT.ModeBit2 := FALSE;
   STATUS[369].EXT.ModeBit3 := FALSE;
   STATUS[369].EXT.BIT19 := FALSE;
   STATUS[369].EXT.BIT20 := FALSE;
   STATUS[369].EXT.AlarmSuppressed := FALSE;
   STATUS[369].EXT.AlarmPrsent := FALSE;
   STATUS[369].EXT.AlarmFailUnAck := FALSE;
   STATUS[369].Status := 0;
   STATUS[369].TimeStamp := 16#0000;
   STATUS[370].VALUE := 0.0;
   STATUS[370].TRIGVALUE := 0.0;
   STATUS[370].EXT.AlarmWarnUnAck := FALSE;
   STATUS[370].EXT.AckRequired := FALSE;
   STATUS[370].EXT.Maintanence := FALSE;
   STATUS[370].EXT.Operation := FALSE;
   STATUS[370].EXT.Forced := FALSE;
   STATUS[370].EXT.BIT29 := FALSE;
   STATUS[370].EXT.BIT30 := FALSE;
   STATUS[370].EXT.BIT31 := FALSE;
   STATUS[370].EXT.ModeBit1 := FALSE;
   STATUS[370].EXT.ModeBit2 := FALSE;
   STATUS[370].EXT.ModeBit3 := FALSE;
   STATUS[370].EXT.BIT19 := FALSE;
   STATUS[370].EXT.BIT20 := FALSE;
   STATUS[370].EXT.AlarmSuppressed := FALSE;
   STATUS[370].EXT.AlarmPrsent := FALSE;
   STATUS[370].EXT.AlarmFailUnAck := FALSE;
   STATUS[370].Status := 0;
   STATUS[370].TimeStamp := 16#0000;
   STATUS[371].VALUE := 0.0;
   STATUS[371].TRIGVALUE := 0.0;
   STATUS[371].EXT.AlarmWarnUnAck := FALSE;
   STATUS[371].EXT.AckRequired := FALSE;
   STATUS[371].EXT.Maintanence := FALSE;
   STATUS[371].EXT.Operation := FALSE;
   STATUS[371].EXT.Forced := FALSE;
   STATUS[371].EXT.BIT29 := FALSE;
   STATUS[371].EXT.BIT30 := FALSE;
   STATUS[371].EXT.BIT31 := FALSE;
   STATUS[371].EXT.ModeBit1 := FALSE;
   STATUS[371].EXT.ModeBit2 := FALSE;
   STATUS[371].EXT.ModeBit3 := FALSE;
   STATUS[371].EXT.BIT19 := FALSE;
   STATUS[371].EXT.BIT20 := FALSE;
   STATUS[371].EXT.AlarmSuppressed := FALSE;
   STATUS[371].EXT.AlarmPrsent := FALSE;
   STATUS[371].EXT.AlarmFailUnAck := FALSE;
   STATUS[371].Status := 0;
   STATUS[371].TimeStamp := 16#0000;
   STATUS[372].VALUE := 0.0;
   STATUS[372].TRIGVALUE := 0.0;
   STATUS[372].EXT.AlarmWarnUnAck := FALSE;
   STATUS[372].EXT.AckRequired := FALSE;
   STATUS[372].EXT.Maintanence := FALSE;
   STATUS[372].EXT.Operation := FALSE;
   STATUS[372].EXT.Forced := FALSE;
   STATUS[372].EXT.BIT29 := FALSE;
   STATUS[372].EXT.BIT30 := FALSE;
   STATUS[372].EXT.BIT31 := FALSE;
   STATUS[372].EXT.ModeBit1 := FALSE;
   STATUS[372].EXT.ModeBit2 := FALSE;
   STATUS[372].EXT.ModeBit3 := FALSE;
   STATUS[372].EXT.BIT19 := FALSE;
   STATUS[372].EXT.BIT20 := FALSE;
   STATUS[372].EXT.AlarmSuppressed := FALSE;
   STATUS[372].EXT.AlarmPrsent := FALSE;
   STATUS[372].EXT.AlarmFailUnAck := FALSE;
   STATUS[372].Status := 0;
   STATUS[372].TimeStamp := 16#0000;
   STATUS[373].VALUE := 0.0;
   STATUS[373].TRIGVALUE := 0.0;
   STATUS[373].EXT.AlarmWarnUnAck := FALSE;
